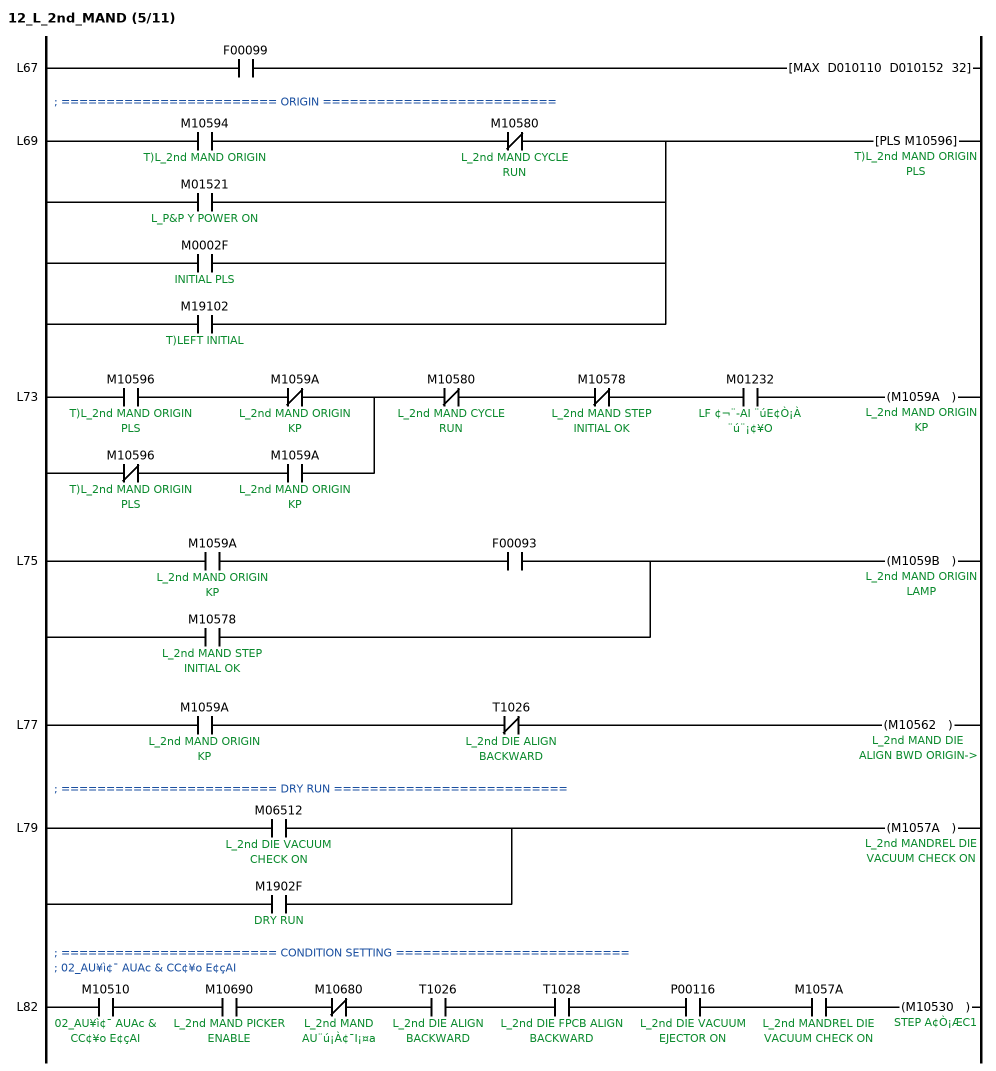
[picture p72: 12_L_2nd_MAND rungs L67-L82]
; L67
LOAD      F00099
MAX       D010110 D010152 32
// ======================== ORIGIN ==========================
; L69
LOAD      M10594	// T)L_2nd MAND ORIGIN
AND NOT   M10580	// L_2nd MAND CYCLE RUN
OR        M01521	// L_P&P Y POWER ON
OR        M0002F	// INITIAL PLS
OR        M19102	// T)LEFT INITIAL
OUTP      M10596	// T)L_2nd MAND ORIGIN PLS
; L73
LOAD      M10596	// T)L_2nd MAND ORIGIN PLS
AND NOT   M1059A	// L_2nd MAND ORIGIN KP
LOAD NOT  M10596	// T)L_2nd MAND ORIGIN PLS
AND       M1059A	// L_2nd MAND ORIGIN KP
OR LOAD
AND NOT   M10580	// L_2nd MAND CYCLE RUN
AND NOT   M10578	// L_2nd MAND STEP INITIAL OK
AND       M01232	// LF ¢¬¨­AI ¨úE¢Ò¡À ¨ú¨¡¢¥O
OUT       M1059A	// L_2nd MAND ORIGIN KP
; L75
LOAD      M1059A	// L_2nd MAND ORIGIN KP
AND       F00093
OR        M10578	// L_2nd MAND STEP INITIAL OK
OUT       M1059B	// L_2nd MAND ORIGIN LAMP
; L77
LOAD      M1059A	// L_2nd MAND ORIGIN KP
AND NOT   T1026	// L_2nd DIE ALIGN BACKWARD
OUT       M10562	// L_2nd MAND DIE ALIGN BWD ORIGIN->
// ======================== DRY RUN ==========================
; L79
LOAD      M06512	// L_2nd DIE VACUUM CHECK ON
OR        M1902F	// DRY RUN
OUT       M1057A	// L_2nd MANDREL DIE VACUUM CHECK ON
// ======================== CONDITION SETTING ==========================
; L82
LOAD      M10510	// 02_AU¥ì¢¯ AUAc & CC¢¥o E¢çAI
AND       M10690	// L_2nd MAND PICKER ENABLE
AND NOT   M10680	// L_2nd MAND AU¨ú¡À¢¯I¡¤a
AND       T1026	// L_2nd DIE ALIGN BACKWARD
AND       T1028	// L_2nd DIE FPCB ALIGN BACKWARD
AND       P00116	// L_2nd DIE VACUUM EJECTOR ON
AND       M1057A	// L_2nd MANDREL DIE VACUUM CHECK ON
OUT       M10530	// STEP A¢Ò¡ÆC1
// output comment: 02_AU¥ì¢¯ AUAc & CC¢¥o E¢çAI

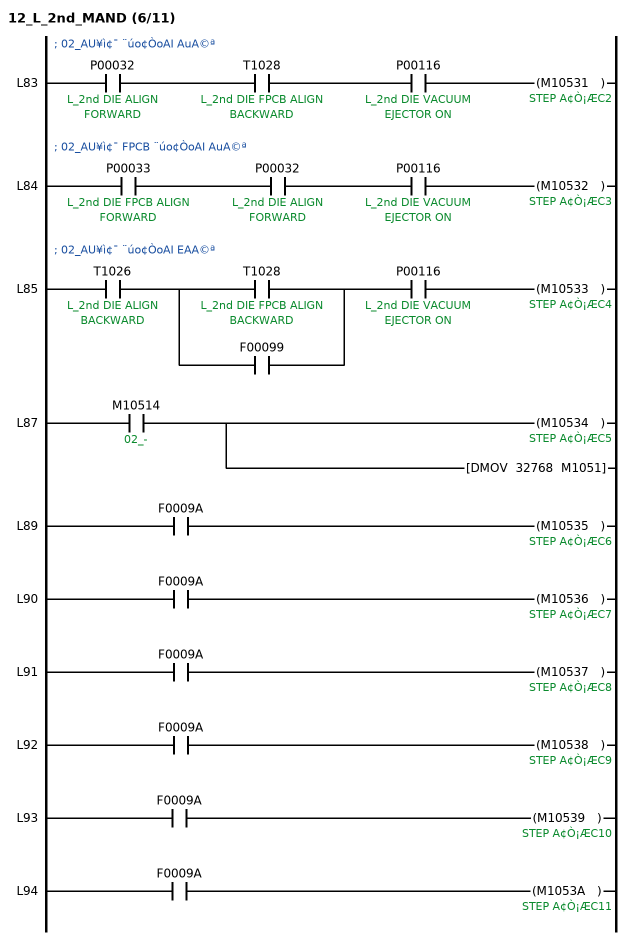
; L83
LOAD      P00032	// L_2nd DIE ALIGN FORWARD
AND       T1028	// L_2nd DIE FPCB ALIGN BACKWARD
AND       P00116	// L_2nd DIE VACUUM EJECTOR ON
OUT       M10531	// STEP A¢Ò¡ÆC2
// output comment: 02_AU¥ì¢¯ ¨úo¢ÒoAI AuA©ª
; L84
LOAD      P00033	// L_2nd DIE FPCB ALIGN FORWARD
AND       P00032	// L_2nd DIE ALIGN FORWARD
AND       P00116	// L_2nd DIE VACUUM EJECTOR ON
OUT       M10532	// STEP A¢Ò¡ÆC3
// output comment: 02_AU¥ì¢¯ FPCB ¨úo¢ÒoAI AuA©ª
; L85
LOAD      T1026	// L_2nd DIE ALIGN BACKWARD
LOAD      T1028	// L_2nd DIE FPCB ALIGN BACKWARD
OR        F00099
AND LOAD
AND       P00116	// L_2nd DIE VACUUM EJECTOR ON
OUT       M10533	// STEP A¢Ò¡ÆC4
// output comment: 02_AU¥ì¢¯ ¨úo¢ÒoAI EAA©ª
; L87
LOAD      M10514	// 02_-
OUT       M10534	// STEP A¢Ò¡ÆC5
DMOV      32768 M1051
; L89
LOAD      F0009A
OUT       M10535	// STEP A¢Ò¡ÆC6
; L90
LOAD      F0009A
OUT       M10536	// STEP A¢Ò¡ÆC7
; L91
LOAD      F0009A
OUT       M10537	// STEP A¢Ò¡ÆC8
; L92
LOAD      F0009A
OUT       M10538	// STEP A¢Ò¡ÆC9
; L93
LOAD      F0009A
OUT       M10539	// STEP A¢Ò¡ÆC10
; L94
LOAD      F0009A
OUT       M1053A	// STEP A¢Ò¡ÆC11

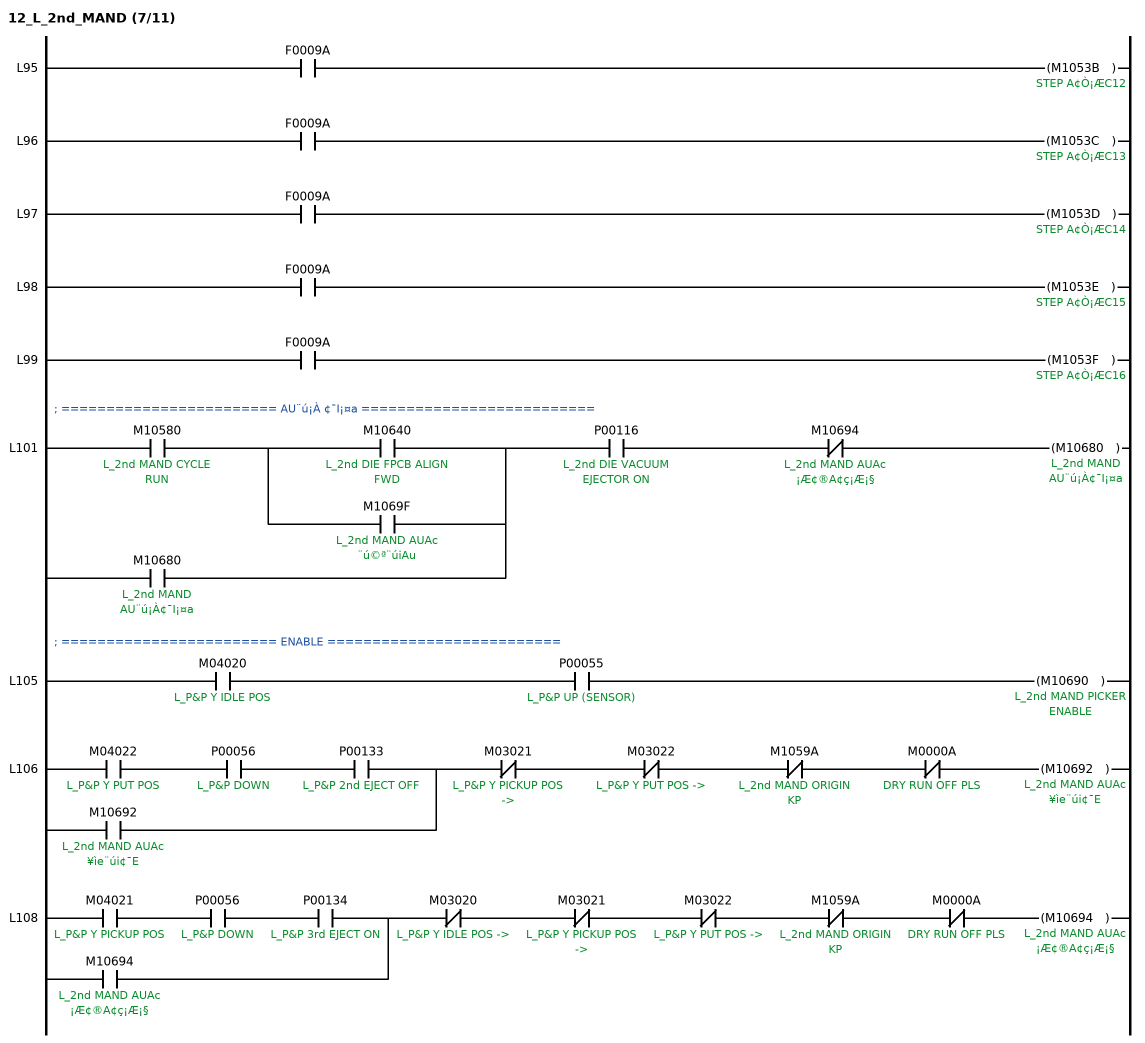
; L95
LOAD      F0009A
OUT       M1053B	// STEP A¢Ò¡ÆC12
; L96
LOAD      F0009A
OUT       M1053C	// STEP A¢Ò¡ÆC13
; L97
LOAD      F0009A
OUT       M1053D	// STEP A¢Ò¡ÆC14
; L98
LOAD      F0009A
OUT       M1053E	// STEP A¢Ò¡ÆC15
; L99
LOAD      F0009A
OUT       M1053F	// STEP A¢Ò¡ÆC16
// ======================== AU¨ú¡À ¢¯I¡¤a ==========================
; L101
LOAD      M10580	// L_2nd MAND CYCLE RUN
LOAD      M10640	// L_2nd DIE FPCB ALIGN FWD
OR        M1069F	// L_2nd MAND AUAc ¨ú©ª¨úiAu
AND LOAD
OR        M10680	// L_2nd MAND AU¨ú¡À¢¯I¡¤a
AND       P00116	// L_2nd DIE VACUUM EJECTOR ON
AND NOT   M10694	// L_2nd MAND AUAc ¡Æ¢®A¢ç¡Æ¡§
OUT       M10680	// L_2nd MAND AU¨ú¡À¢¯I¡¤a
// ======================== ENABLE ==========================
; L105
LOAD      M04020	// L_P&P Y IDLE POS
AND       P00055	// L_P&P UP (SENSOR)
OUT       M10690	// L_2nd MAND PICKER ENABLE
; L106
LOAD      M04022	// L_P&P Y PUT POS
AND       P00056	// L_P&P DOWN
AND       P00133	// L_P&P 2nd EJECT OFF
OR        M10692	// L_2nd MAND AUAc ¥ìe¨úi¢¯E
AND NOT   M03021	// L_P&P Y PICKUP POS ->
AND NOT   M03022	// L_P&P Y PUT POS ->
AND NOT   M1059A	// L_2nd MAND ORIGIN KP
AND NOT   M0000A	// DRY RUN OFF PLS
OUT       M10692	// L_2nd MAND AUAc ¥ìe¨úi¢¯E
; L108
LOAD      M04021	// L_P&P Y PICKUP POS
AND       P00056	// L_P&P DOWN
AND       P00134	// L_P&P 3rd EJECT ON
OR        M10694	// L_2nd MAND AUAc ¡Æ¢®A¢ç¡Æ¡§
AND NOT   M03020	// L_P&P Y IDLE POS ->
AND NOT   M03021	// L_P&P Y PICKUP POS ->
AND NOT   M03022	// L_P&P Y PUT POS ->
AND NOT   M1059A	// L_2nd MAND ORIGIN KP
AND NOT   M0000A	// DRY RUN OFF PLS
OUT       M10694	// L_2nd MAND AUAc ¡Æ¢®A¢ç¡Æ¡§

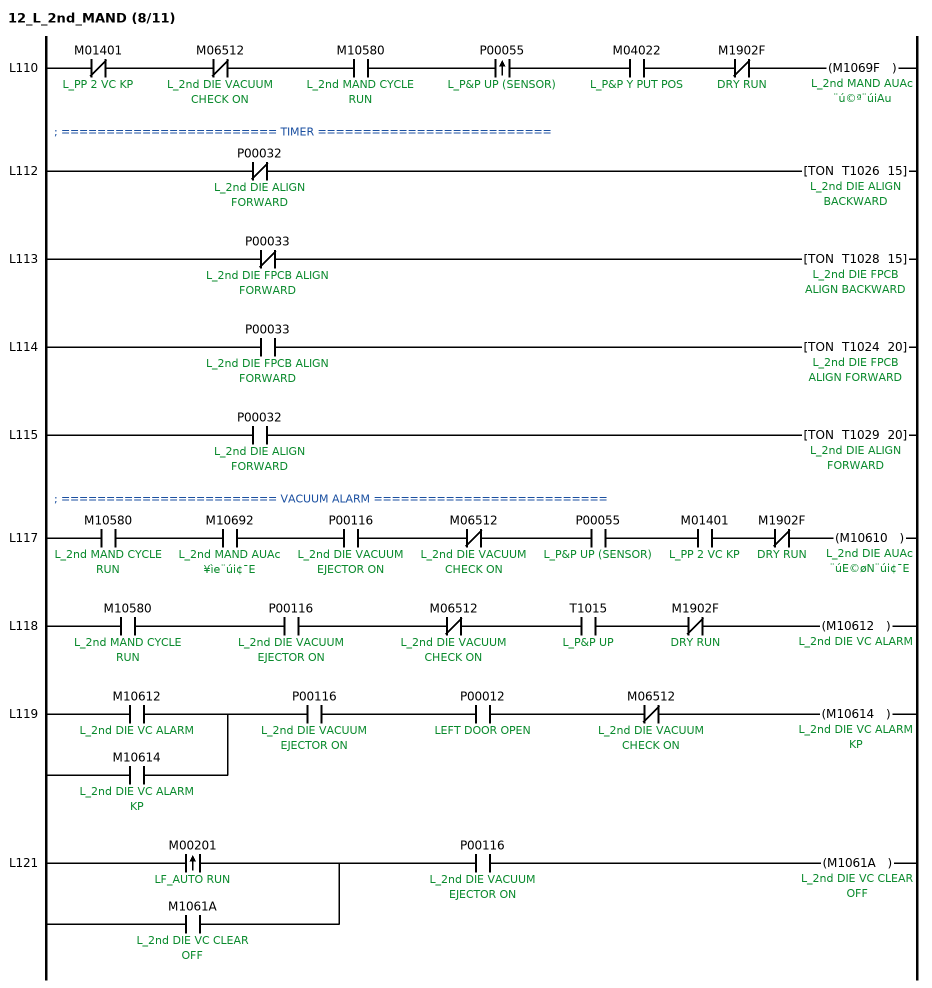
; L110
LOAD NOT  M01401	// L_PP 2 VC KP
AND NOT   M06512	// L_2nd DIE VACUUM CHECK ON
AND       M10580	// L_2nd MAND CYCLE RUN
ANDP      P00055	// L_P&P UP (SENSOR)
AND       M04022	// L_P&P Y PUT POS
AND NOT   M1902F	// DRY RUN
OUT       M1069F	// L_2nd MAND AUAc ¨ú©ª¨úiAu
// ======================== TIMER ==========================
; L112
LOAD NOT  P00032	// L_2nd DIE ALIGN FORWARD
TON       T1026 15	// L_2nd DIE ALIGN BACKWARD
; L113
LOAD NOT  P00033	// L_2nd DIE FPCB ALIGN FORWARD
TON       T1028 15	// L_2nd DIE FPCB ALIGN BACKWARD
; L114
LOAD      P00033	// L_2nd DIE FPCB ALIGN FORWARD
TON       T1024 20	// L_2nd DIE FPCB ALIGN FORWARD
; L115
LOAD      P00032	// L_2nd DIE ALIGN FORWARD
TON       T1029 20	// L_2nd DIE ALIGN FORWARD
// ======================== VACUUM ALARM ==========================
; L117
LOAD      M10580	// L_2nd MAND CYCLE RUN
AND       M10692	// L_2nd MAND AUAc ¥ìe¨úi¢¯E
AND       P00116	// L_2nd DIE VACUUM EJECTOR ON
AND NOT   M06512	// L_2nd DIE VACUUM CHECK ON
AND       P00055	// L_P&P UP (SENSOR)
AND       M01401	// L_PP 2 VC KP
AND NOT   M1902F	// DRY RUN
OUT       M10610	// L_2nd DIE AUAc ¨úE©øN¨úi¢¯E
; L118
LOAD      M10580	// L_2nd MAND CYCLE RUN
AND       P00116	// L_2nd DIE VACUUM EJECTOR ON
AND NOT   M06512	// L_2nd DIE VACUUM CHECK ON
AND       T1015	// L_P&P UP
AND NOT   M1902F	// DRY RUN
OUT       M10612	// L_2nd DIE VC ALARM
; L119
LOAD      M10612	// L_2nd DIE VC ALARM
OR        M10614	// L_2nd DIE VC ALARM KP
AND       P00116	// L_2nd DIE VACUUM EJECTOR ON
AND       P00012	// LEFT DOOR OPEN
AND NOT   M06512	// L_2nd DIE VACUUM CHECK ON
OUT       M10614	// L_2nd DIE VC ALARM KP
; L121
LOADP     M00201	// LF_AUTO RUN
OR        M1061A	// L_2nd DIE VC CLEAR OFF
AND       P00116	// L_2nd DIE VACUUM EJECTOR ON
OUT       M1061A	// L_2nd DIE VC CLEAR OFF

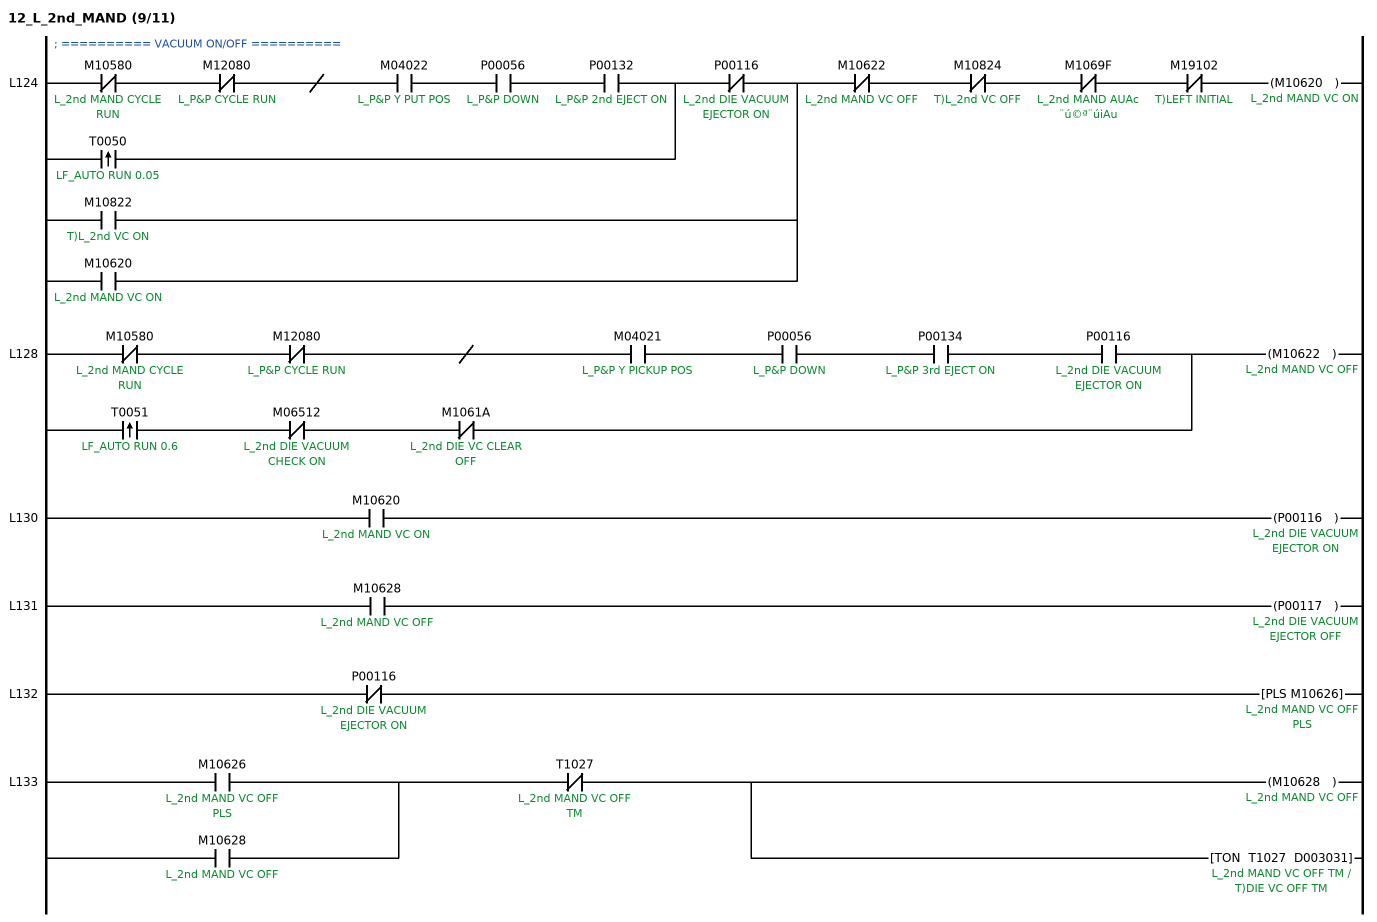
// ========== VACUUM ON/OFF ==========
; L124
LOAD NOT  M10580	// L_2nd MAND CYCLE RUN
AND NOT   M12080	// L_P&P CYCLE RUN
NOT
AND       M04022	// L_P&P Y PUT POS
AND       P00056	// L_P&P DOWN
AND       P00132	// L_P&P 2nd EJECT ON
ORP       T0050	// LF_AUTO RUN 0.05
AND NOT   P00116	// L_2nd DIE VACUUM EJECTOR ON
OR        M10822	// T)L_2nd VC ON
OR        M10620	// L_2nd MAND VC ON
AND NOT   M10622	// L_2nd MAND VC OFF
AND NOT   M10824	// T)L_2nd VC OFF
AND NOT   M1069F	// L_2nd MAND AUAc ¨ú©ª¨úiAu
AND NOT   M19102	// T)LEFT INITIAL
OUT       M10620	// L_2nd MAND VC ON
; L128
LOAD NOT  M10580	// L_2nd MAND CYCLE RUN
AND NOT   M12080	// L_P&P CYCLE RUN
NOT
AND       M04021	// L_P&P Y PICKUP POS
AND       P00056	// L_P&P DOWN
AND       P00134	// L_P&P 3rd EJECT ON
AND       P00116	// L_2nd DIE VACUUM EJECTOR ON
LOADP     T0051	// LF_AUTO RUN 0.6
AND NOT   M06512	// L_2nd DIE VACUUM CHECK ON
AND NOT   M1061A	// L_2nd DIE VC CLEAR OFF
OR LOAD
OUT       M10622	// L_2nd MAND VC OFF
; L130
LOAD      M10620	// L_2nd MAND VC ON
OUT       P00116	// L_2nd DIE VACUUM EJECTOR ON
; L131
LOAD      M10628	// L_2nd MAND VC OFF
OUT       P00117	// L_2nd DIE VACUUM EJECTOR OFF
; L132
LOAD NOT  P00116	// L_2nd DIE VACUUM EJECTOR ON
OUTP      M10626	// L_2nd MAND VC OFF PLS
; L133
LOAD      M10626	// L_2nd MAND VC OFF PLS
OR        M10628	// L_2nd MAND VC OFF
AND NOT   T1027	// L_2nd MAND VC OFF TM
OUT       M10628	// L_2nd MAND VC OFF
TON       T1027 D003031	// L_2nd MAND VC OFF TM / T)DIE VC OFF TM

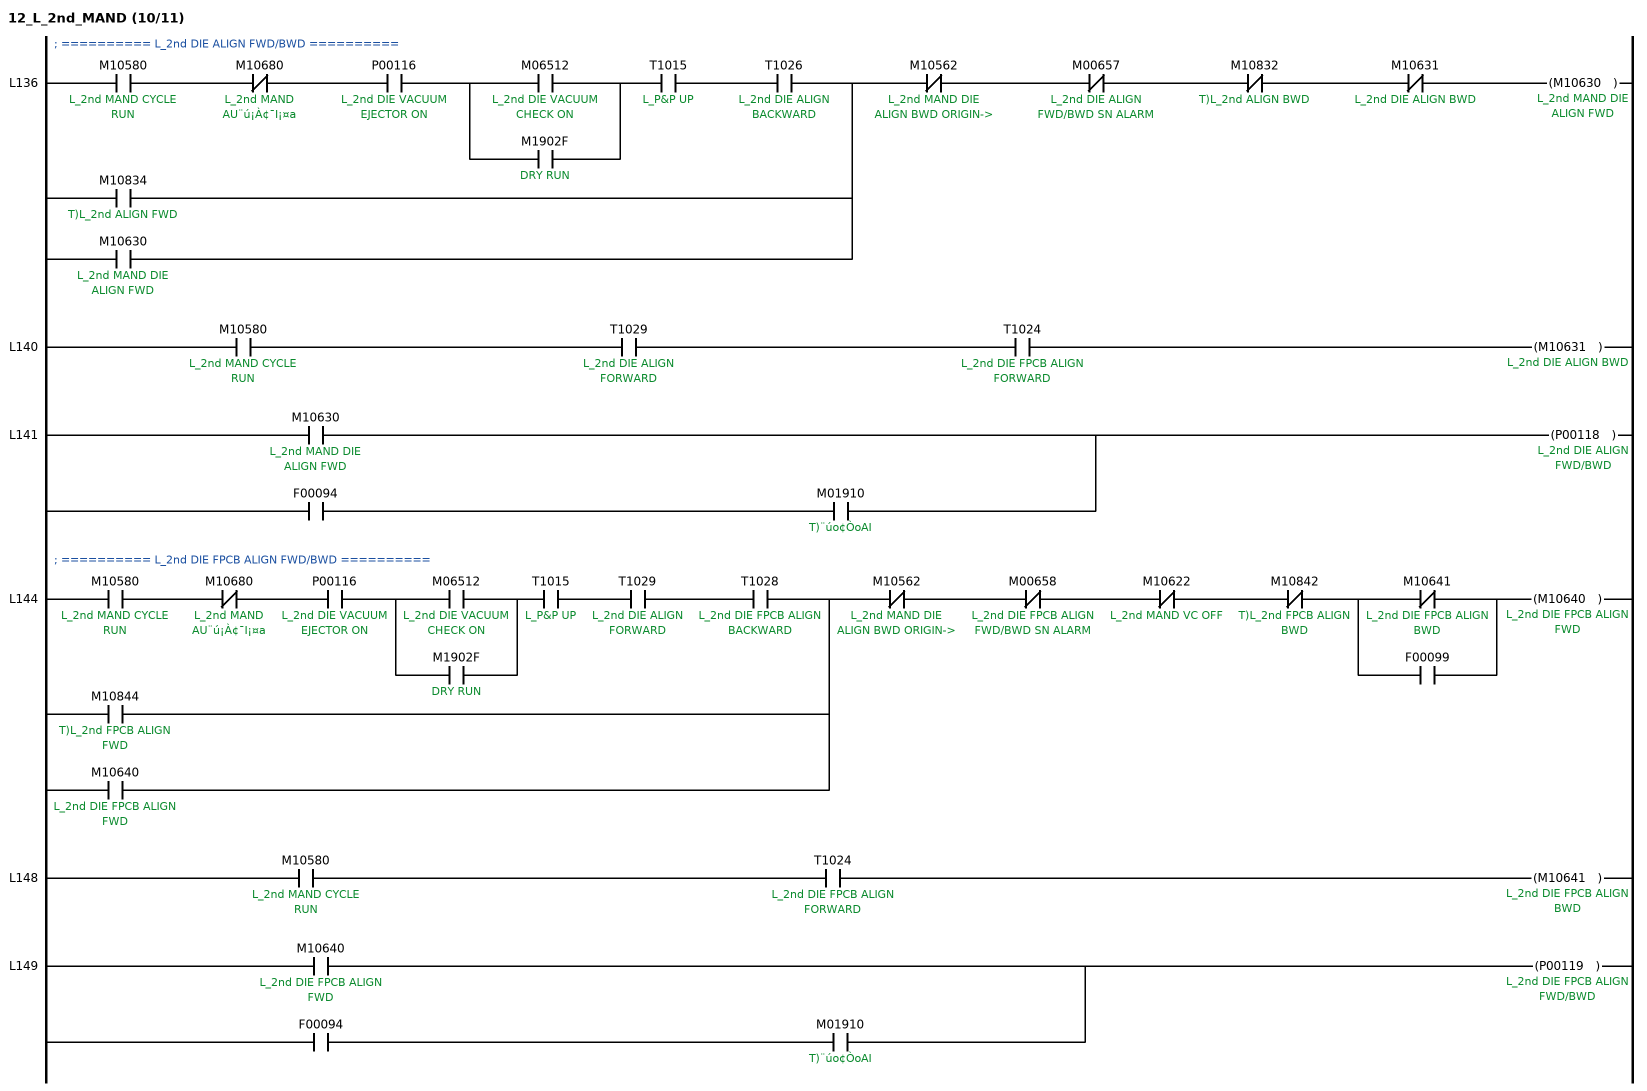
// ========== L_2nd DIE ALIGN FWD/BWD ==========
; L136
LOAD      M10580	// L_2nd MAND CYCLE RUN
AND NOT   M10680	// L_2nd MAND AU¨ú¡À¢¯I¡¤a
AND       P00116	// L_2nd DIE VACUUM EJECTOR ON
LOAD      M06512	// L_2nd DIE VACUUM CHECK ON
OR        M1902F	// DRY RUN
AND LOAD
AND       T1015	// L_P&P UP
AND       T1026	// L_2nd DIE ALIGN BACKWARD
OR        M10834	// T)L_2nd ALIGN FWD
OR        M10630	// L_2nd MAND DIE ALIGN FWD
AND NOT   M10562	// L_2nd MAND DIE ALIGN BWD ORIGIN->
AND NOT   M00657	// L_2nd DIE ALIGN FWD/BWD SN ALARM
AND NOT   M10832	// T)L_2nd ALIGN BWD
AND NOT   M10631	// L_2nd DIE ALIGN BWD
OUT       M10630	// L_2nd MAND DIE ALIGN FWD
; L140
LOAD      M10580	// L_2nd MAND CYCLE RUN
AND       T1029	// L_2nd DIE ALIGN FORWARD
AND       T1024	// L_2nd DIE FPCB ALIGN FORWARD
OUT       M10631	// L_2nd DIE ALIGN BWD
; L141
LOAD      M10630	// L_2nd MAND DIE ALIGN FWD
LOAD      F00094
AND       M01910	// T)¨úo¢ÒoAI
OR LOAD
OUT       P00118	// L_2nd DIE ALIGN FWD/BWD
// ========== L_2nd DIE FPCB ALIGN FWD/BWD ==========
; L144
LOAD      M10580	// L_2nd MAND CYCLE RUN
AND NOT   M10680	// L_2nd MAND AU¨ú¡À¢¯I¡¤a
AND       P00116	// L_2nd DIE VACUUM EJECTOR ON
LOAD      M06512	// L_2nd DIE VACUUM CHECK ON
OR        M1902F	// DRY RUN
AND LOAD
AND       T1015	// L_P&P UP
AND       T1029	// L_2nd DIE ALIGN FORWARD
AND       T1028	// L_2nd DIE FPCB ALIGN BACKWARD
OR        M10844	// T)L_2nd FPCB ALIGN FWD
OR        M10640	// L_2nd DIE FPCB ALIGN FWD
AND NOT   M10562	// L_2nd MAND DIE ALIGN BWD ORIGIN->
AND NOT   M00658	// L_2nd DIE FPCB ALIGN FWD/BWD SN ALARM
AND NOT   M10622	// L_2nd MAND VC OFF
AND NOT   M10842	// T)L_2nd FPCB ALIGN BWD
LOAD NOT  M10641	// L_2nd DIE FPCB ALIGN BWD
OR        F00099
AND LOAD
OUT       M10640	// L_2nd DIE FPCB ALIGN FWD
; L148
LOAD      M10580	// L_2nd MAND CYCLE RUN
AND       T1024	// L_2nd DIE FPCB ALIGN FORWARD
OUT       M10641	// L_2nd DIE FPCB ALIGN BWD
; L149
LOAD      M10640	// L_2nd DIE FPCB ALIGN FWD
LOAD      F00094
AND       M01910	// T)¨úo¢ÒoAI
OR LOAD
OUT       P00119	// L_2nd DIE FPCB ALIGN FWD/BWD

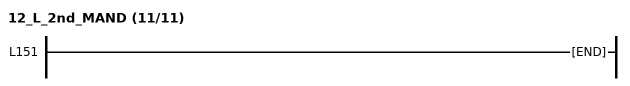
; L151
END

PROGRAM 13_L_3rd_MAND (task: ¨ö¨¬A¥ì CA¡¤I¡¾¡¿¡¤¡Í)

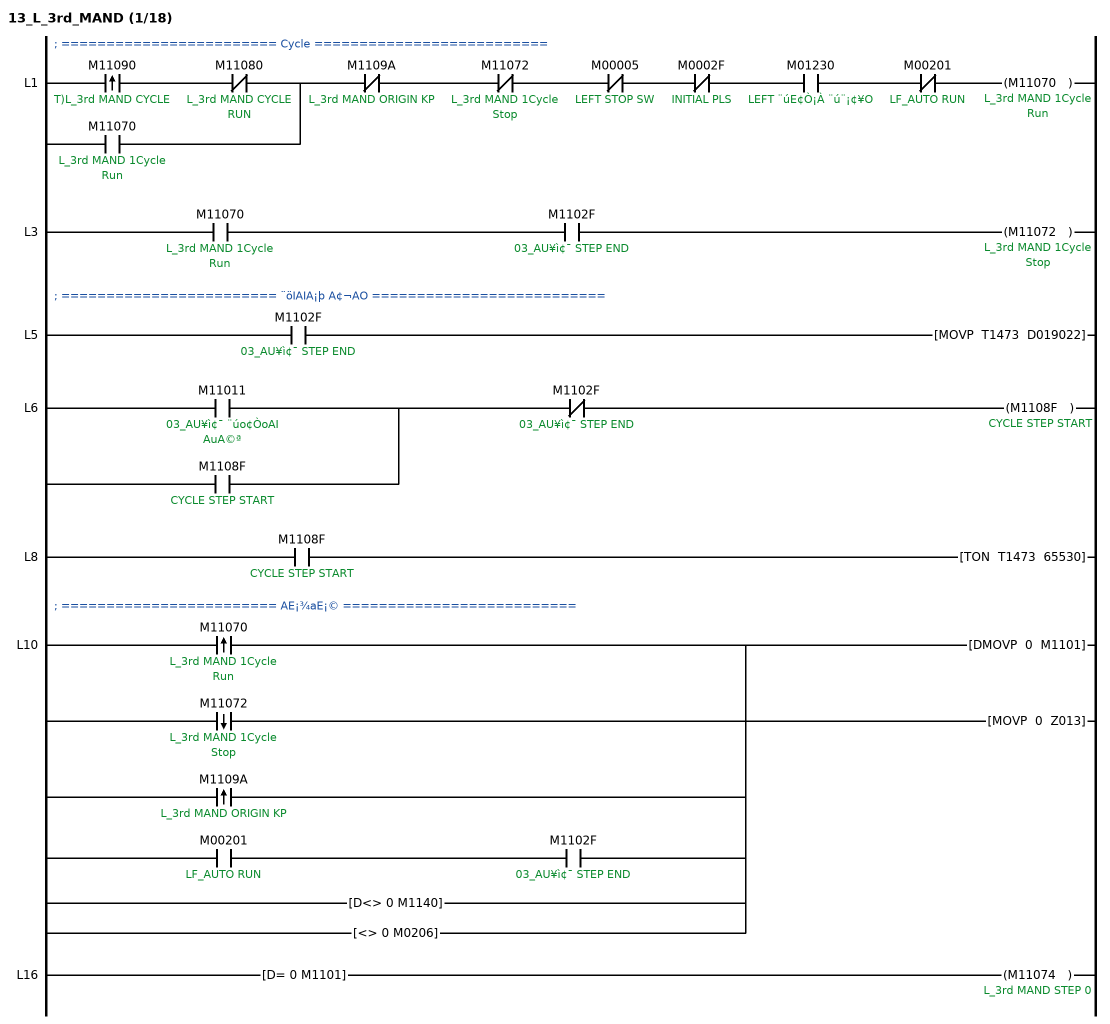
// ======================== Cycle ==========================
; L1
LOADP     M11090	// T)L_3rd MAND CYCLE
AND NOT   M11080	// L_3rd MAND CYCLE RUN
OR        M11070	// L_3rd MAND 1Cycle Run
AND NOT   M1109A	// L_3rd MAND ORIGIN KP
AND NOT   M11072	// L_3rd MAND 1Cycle Stop
AND NOT   M00005	// LEFT STOP SW
AND NOT   M0002F	// INITIAL PLS
AND       M01230	// LEFT ¨úE¢Ò¡À ¨ú¨¡¢¥O
AND NOT   M00201	// LF_AUTO RUN
OUT       M11070	// L_3rd MAND 1Cycle Run
; L3
LOAD      M11070	// L_3rd MAND 1Cycle Run
AND       M1102F	// 03_AU¥ì¢¯ STEP END
OUT       M11072	// L_3rd MAND 1Cycle Stop
// ======================== ¨öIAIA¡þ A¢¬AO ==========================
; L5
LOAD      M1102F	// 03_AU¥ì¢¯ STEP END
MOVP      T1473 D019022
; L6
LOAD      M11011	// 03_AU¥ì¢¯ ¨úo¢ÒoAI AuA©ª
OR        M1108F	// CYCLE STEP START
AND NOT   M1102F	// 03_AU¥ì¢¯ STEP END
OUT       M1108F	// CYCLE STEP START
; L8
LOAD      M1108F	// CYCLE STEP START
TON       T1473 65530
// ======================== AE¡¾aE¡© ==========================
; L10
LOADP     M11070	// L_3rd MAND 1Cycle Run
ORN       M11072	// L_3rd MAND 1Cycle Stop
ORP       M1109A	// L_3rd MAND ORIGIN KP
LOAD      M00201	// LF_AUTO RUN
AND       M1102F	// 03_AU¥ì¢¯ STEP END
OR LOAD
ORD<>     0 M1140
OR<>      0 M0206
DMOVP     0 M1101
MOVP      0 Z013
; L16
LOADD=    0 M1101
OUT       M11074	// L_3rd MAND STEP 0

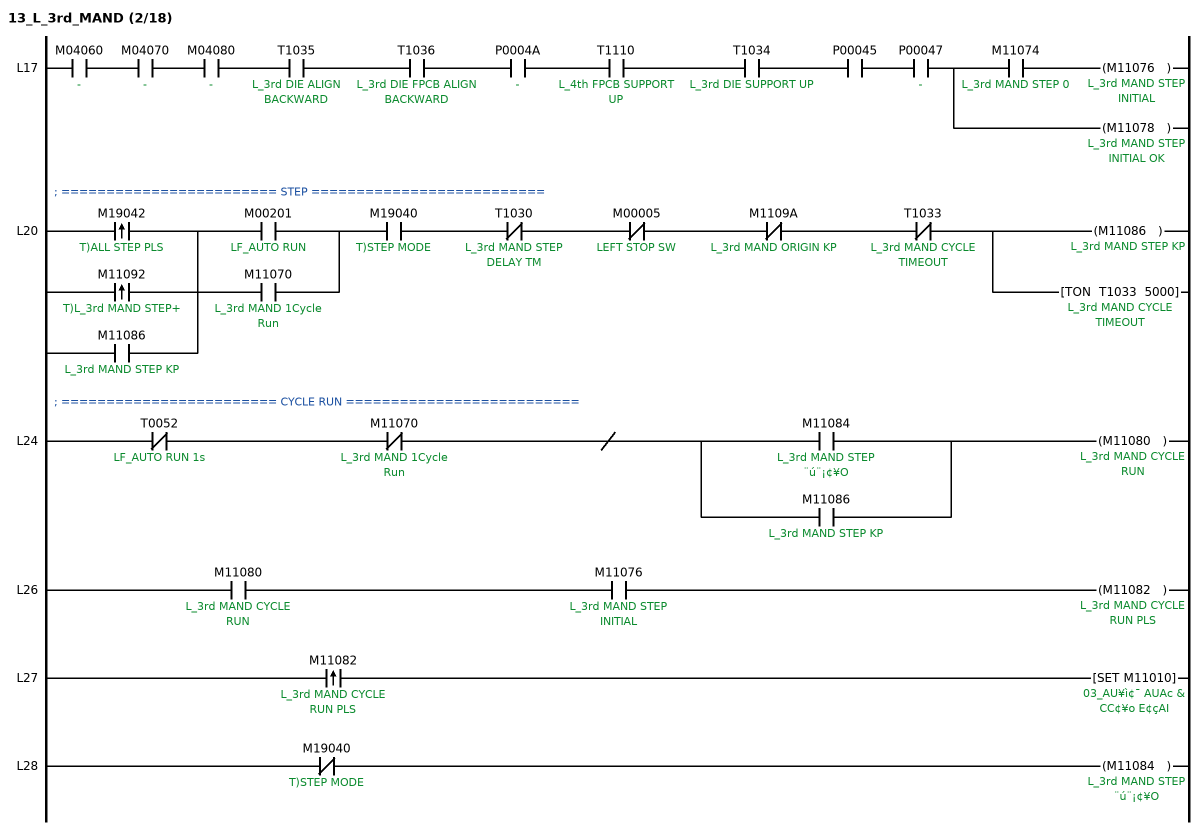
; L17
LOAD      M04060	// -
AND       M04070	// -
AND       M04080	// -
AND       T1035	// L_3rd DIE ALIGN BACKWARD
AND       T1036	// L_3rd DIE FPCB ALIGN BACKWARD
AND       P0004A	// -
AND       T1110	// L_4th FPCB SUPPORT UP
AND       T1034	// L_3rd DIE SUPPORT UP
AND       P00045
AND       P00047	// -
MPUSH
AND       M11074	// L_3rd MAND STEP 0
OUT       M11076	// L_3rd MAND STEP INITIAL
MPOP
OUT       M11078	// L_3rd MAND STEP INITIAL OK
// ======================== STEP ==========================
; L20
LOADP     M19042	// T)ALL STEP PLS
ORP       M11092	// T)L_3rd MAND STEP+
OR        M11086	// L_3rd MAND STEP KP
LOAD      M00201	// LF_AUTO RUN
OR        M11070	// L_3rd MAND 1Cycle Run
AND LOAD
AND       M19040	// T)STEP MODE
AND NOT   T1030	// L_3rd MAND STEP DELAY TM
AND NOT   M00005	// LEFT STOP SW
AND NOT   M1109A	// L_3rd MAND ORIGIN KP
AND NOT   T1033	// L_3rd MAND CYCLE TIMEOUT
OUT       M11086	// L_3rd MAND STEP KP
TON       T1033 5000	// L_3rd MAND CYCLE TIMEOUT
// ======================== CYCLE RUN ==========================
; L24
LOAD NOT  T0052	// LF_AUTO RUN 1s
AND NOT   M11070	// L_3rd MAND 1Cycle Run
NOT
LOAD      M11084	// L_3rd MAND STEP ¨ú¨¡¢¥O
OR        M11086	// L_3rd MAND STEP KP
AND LOAD
OUT       M11080	// L_3rd MAND CYCLE RUN
; L26
LOAD      M11080	// L_3rd MAND CYCLE RUN
AND       M11076	// L_3rd MAND STEP INITIAL
OUT       M11082	// L_3rd MAND CYCLE RUN PLS
; L27
LOADP     M11082	// L_3rd MAND CYCLE RUN PLS
SET       M11010	// 03_AU¥ì¢¯ AUAc & CC¢¥o E¢çAI
; L28
LOAD NOT  M19040	// T)STEP MODE
OUT       M11084	// L_3rd MAND STEP ¨ú¨¡¢¥O

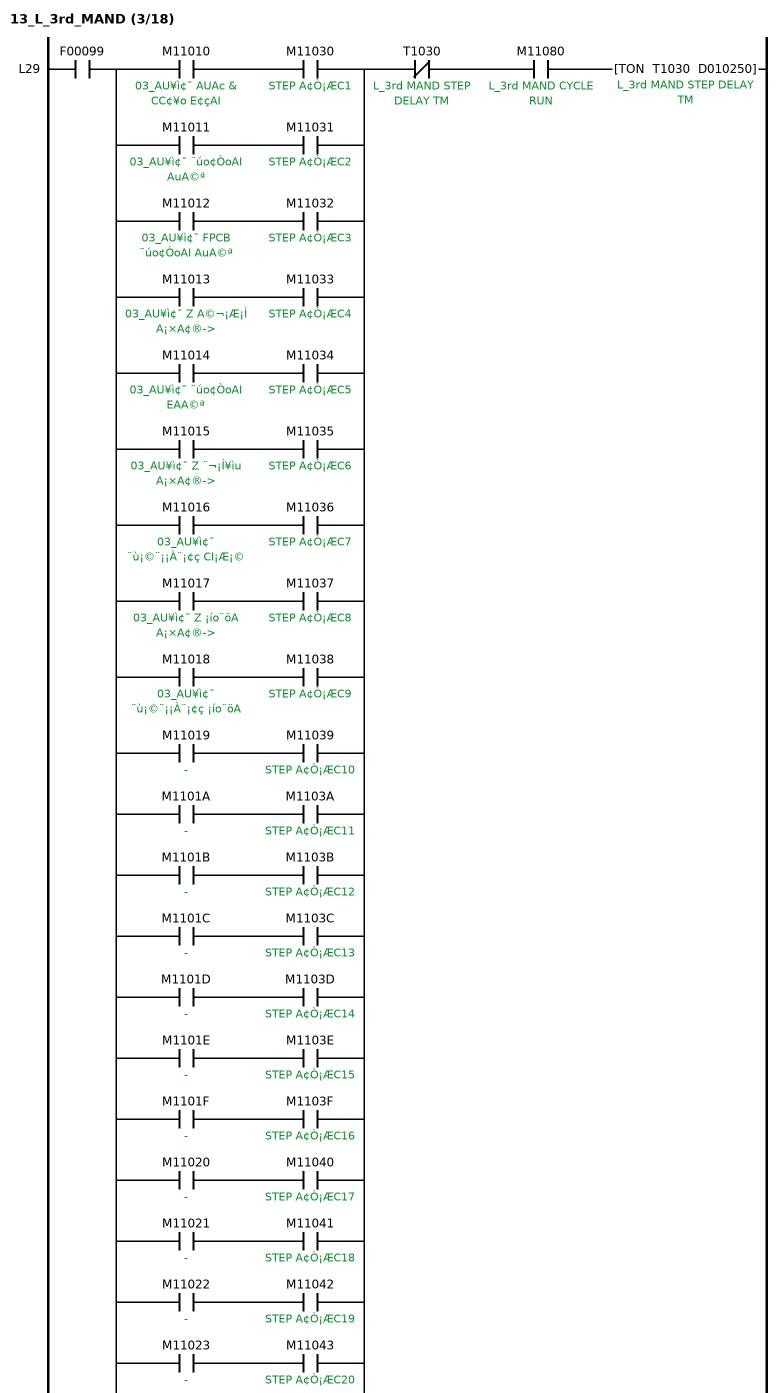

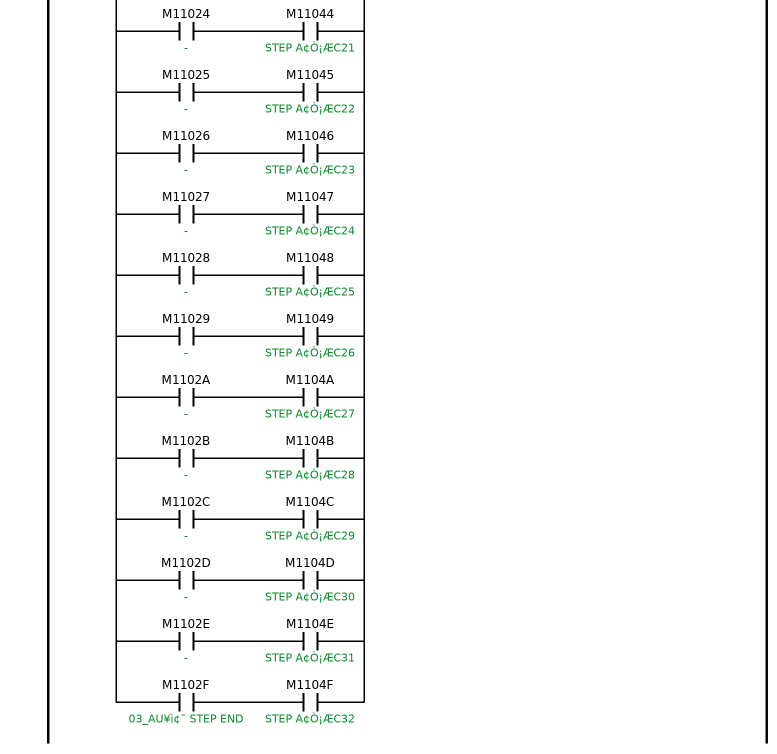
; L29
LOAD      F00099
LOAD      M11010	// 03_AU¥ì¢¯ AUAc & CC¢¥o E¢çAI
AND       M11030	// STEP A¢Ò¡ÆC1
LOAD      M11011	// 03_AU¥ì¢¯ ¨úo¢ÒoAI AuA©ª
AND       M11031	// STEP A¢Ò¡ÆC2
OR LOAD
LOAD      M11012	// 03_AU¥ì¢¯ FPCB ¨úo¢ÒoAI AuA©ª
AND       M11032	// STEP A¢Ò¡ÆC3
OR LOAD
LOAD      M11013	// 03_AU¥ì¢¯ Z A©¬¡Æ¡Ì A¡×A¢®->
AND       M11033	// STEP A¢Ò¡ÆC4
OR LOAD
LOAD      M11014	// 03_AU¥ì¢¯ ¨úo¢ÒoAI EAA©ª
AND       M11034	// STEP A¢Ò¡ÆC5
OR LOAD
LOAD      M11015	// 03_AU¥ì¢¯ Z ¨¬¡Í¥ìu A¡×A¢®->
AND       M11035	// STEP A¢Ò¡ÆC6
OR LOAD
LOAD      M11016	// 03_AU¥ì¢¯ ¨ù¡©¨¡¡À¨¡¢ç CI¡Æ¡©
AND       M11036	// STEP A¢Ò¡ÆC7
OR LOAD
LOAD      M11017	// 03_AU¥ì¢¯ Z ¡ío¨öA A¡×A¢®->
AND       M11037	// STEP A¢Ò¡ÆC8
OR LOAD
LOAD      M11018	// 03_AU¥ì¢¯ ¨ù¡©¨¡¡À¨¡¢ç ¡ío¨öA
AND       M11038	// STEP A¢Ò¡ÆC9
OR LOAD
LOAD      M11019	// -
AND       M11039	// STEP A¢Ò¡ÆC10
OR LOAD
LOAD      M1101A	// -
AND       M1103A	// STEP A¢Ò¡ÆC11
OR LOAD
LOAD      M1101B	// -
AND       M1103B	// STEP A¢Ò¡ÆC12
OR LOAD
LOAD      M1101C	// -
AND       M1103C	// STEP A¢Ò¡ÆC13
OR LOAD
LOAD      M1101D	// -
AND       M1103D	// STEP A¢Ò¡ÆC14
OR LOAD
LOAD      M1101E	// -
AND       M1103E	// STEP A¢Ò¡ÆC15
OR LOAD
LOAD      M1101F	// -
AND       M1103F	// STEP A¢Ò¡ÆC16
OR LOAD
LOAD      M11020	// -
AND       M11040	// STEP A¢Ò¡ÆC17
OR LOAD
LOAD      M11021	// -
AND       M11041	// STEP A¢Ò¡ÆC18
OR LOAD
LOAD      M11022	// -
AND       M11042	// STEP A¢Ò¡ÆC19
OR LOAD
LOAD      M11023	// -
AND       M11043	// STEP A¢Ò¡ÆC20
OR LOAD
LOAD      M11024	// -
AND       M11044	// STEP A¢Ò¡ÆC21
OR LOAD
LOAD      M11025	// -
AND       M11045	// STEP A¢Ò¡ÆC22
OR LOAD
LOAD      M11026	// -
AND       M11046	// STEP A¢Ò¡ÆC23
OR LOAD
LOAD      M11027	// -
AND       M11047	// STEP A¢Ò¡ÆC24
OR LOAD
LOAD      M11028	// -
AND       M11048	// STEP A¢Ò¡ÆC25
OR LOAD
LOAD      M11029	// -
AND       M11049	// STEP A¢Ò¡ÆC26
OR LOAD
LOAD      M1102A	// -
AND       M1104A	// STEP A¢Ò¡ÆC27
OR LOAD
LOAD      M1102B	// -
AND       M1104B	// STEP A¢Ò¡ÆC28
OR LOAD
LOAD      M1102C	// -
AND       M1104C	// STEP A¢Ò¡ÆC29
OR LOAD
LOAD      M1102D	// -
AND       M1104D	// STEP A¢Ò¡ÆC30
OR LOAD
LOAD      M1102E	// -
AND       M1104E	// STEP A¢Ò¡ÆC31
OR LOAD
LOAD      M1102F	// 03_AU¥ì¢¯ STEP END
AND       M1104F	// STEP A¢Ò¡ÆC32
OR LOAD
AND LOAD
AND NOT   T1030	// L_3rd MAND STEP DELAY TM
AND       M11080	// L_3rd MAND CYCLE RUN
TON       T1030 D010250	// L_3rd MAND STEP DELAY TM

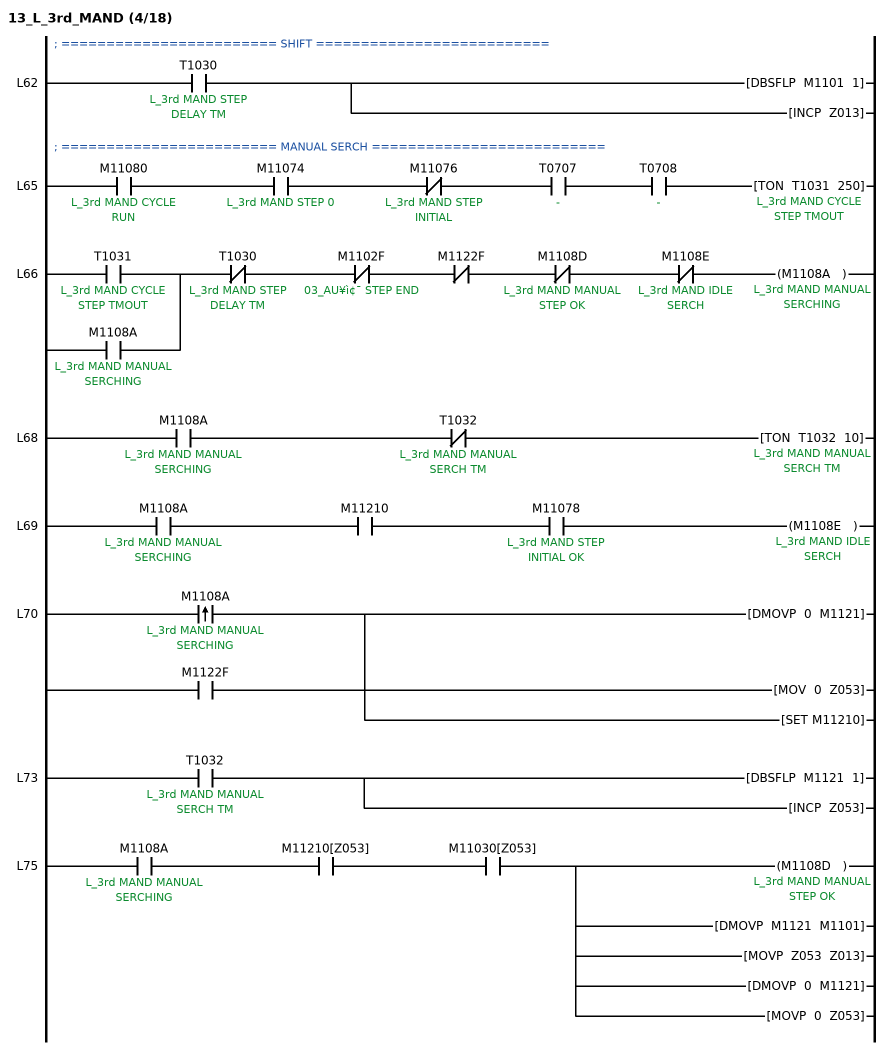
// ======================== SHIFT ==========================
; L62
LOAD      T1030	// L_3rd MAND STEP DELAY TM
DBSFLP    M1101 1
INCP      Z013
// ======================== MANUAL SERCH ==========================
; L65
LOAD      M11080	// L_3rd MAND CYCLE RUN
AND       M11074	// L_3rd MAND STEP 0
AND NOT   M11076	// L_3rd MAND STEP INITIAL
AND       T0707	// -
AND       T0708	// -
TON       T1031 250	// L_3rd MAND CYCLE STEP TMOUT
; L66
LOAD      T1031	// L_3rd MAND CYCLE STEP TMOUT
OR        M1108A	// L_3rd MAND MANUAL SERCHING
AND NOT   T1030	// L_3rd MAND STEP DELAY TM
AND NOT   M1102F	// 03_AU¥ì¢¯ STEP END
AND NOT   M1122F
AND NOT   M1108D	// L_3rd MAND MANUAL STEP OK
AND NOT   M1108E	// L_3rd MAND IDLE SERCH
OUT       M1108A	// L_3rd MAND MANUAL SERCHING
; L68
LOAD      M1108A	// L_3rd MAND MANUAL SERCHING
AND NOT   T1032	// L_3rd MAND MANUAL SERCH TM
TON       T1032 10	// L_3rd MAND MANUAL SERCH TM
; L69
LOAD      M1108A	// L_3rd MAND MANUAL SERCHING
AND       M11210
AND       M11078	// L_3rd MAND STEP INITIAL OK
OUT       M1108E	// L_3rd MAND IDLE SERCH
; L70
LOADP     M1108A	// L_3rd MAND MANUAL SERCHING
OR        M1122F
DMOVP     0 M1121
MOV       0 Z053
SET       M11210
; L73
LOAD      T1032	// L_3rd MAND MANUAL SERCH TM
DBSFLP    M1121 1
INCP      Z053
; L75
LOAD      M1108A	// L_3rd MAND MANUAL SERCHING
AND       M11210[Z053]
AND       M11030[Z053]
OUT       M1108D	// L_3rd MAND MANUAL STEP OK
DMOVP     M1121 M1101
MOVP      Z053 Z013
DMOVP     0 M1121
MOVP      0 Z053

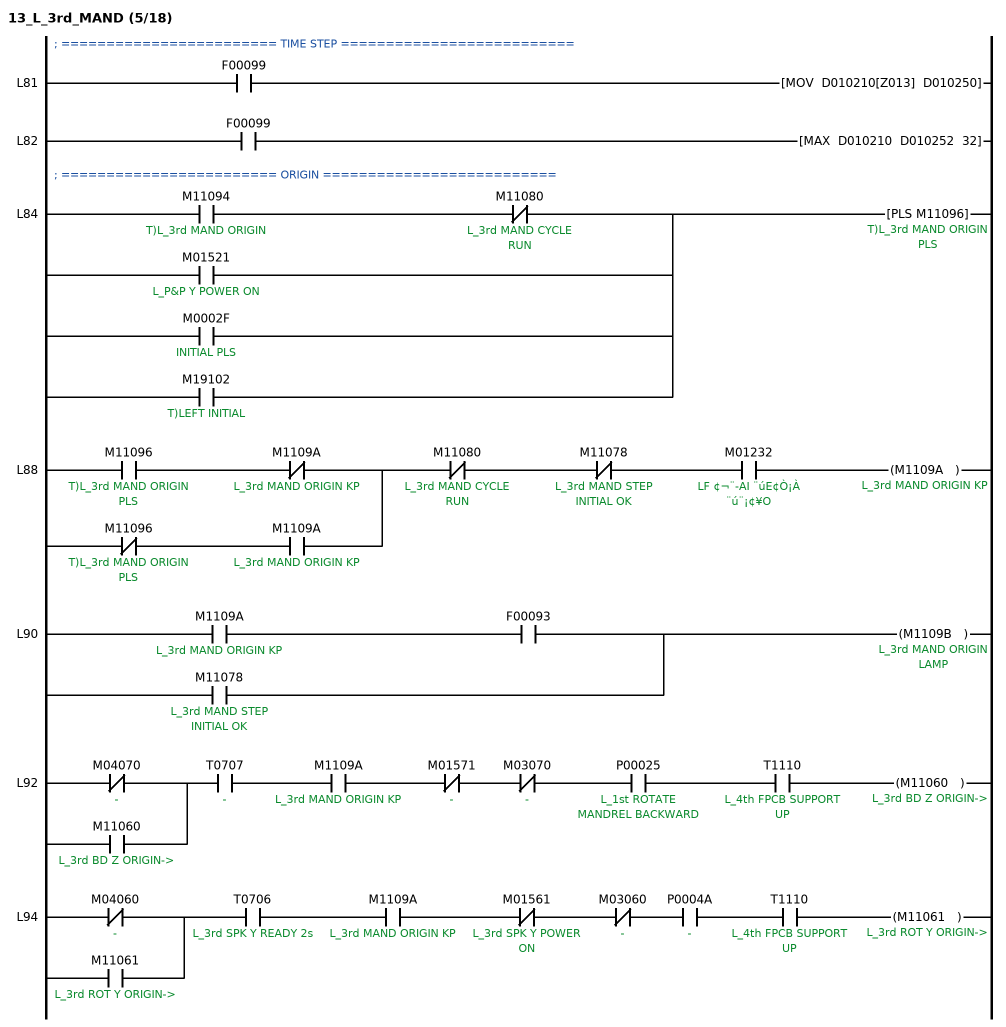
// ======================== TIME STEP ==========================
; L81
LOAD      F00099
MOV       D010210[Z013] D010250
; L82
LOAD      F00099
MAX       D010210 D010252 32
// ======================== ORIGIN ==========================
; L84
LOAD      M11094	// T)L_3rd MAND ORIGIN
AND NOT   M11080	// L_3rd MAND CYCLE RUN
OR        M01521	// L_P&P Y POWER ON
OR        M0002F	// INITIAL PLS
OR        M19102	// T)LEFT INITIAL
OUTP      M11096	// T)L_3rd MAND ORIGIN PLS
; L88
LOAD      M11096	// T)L_3rd MAND ORIGIN PLS
AND NOT   M1109A	// L_3rd MAND ORIGIN KP
LOAD NOT  M11096	// T)L_3rd MAND ORIGIN PLS
AND       M1109A	// L_3rd MAND ORIGIN KP
OR LOAD
AND NOT   M11080	// L_3rd MAND CYCLE RUN
AND NOT   M11078	// L_3rd MAND STEP INITIAL OK
AND       M01232	// LF ¢¬¨­AI ¨úE¢Ò¡À ¨ú¨¡¢¥O
OUT       M1109A	// L_3rd MAND ORIGIN KP
; L90
LOAD      M1109A	// L_3rd MAND ORIGIN KP
AND       F00093
OR        M11078	// L_3rd MAND STEP INITIAL OK
OUT       M1109B	// L_3rd MAND ORIGIN LAMP
; L92
LOAD NOT  M04070	// -
OR        M11060	// L_3rd BD Z ORIGIN->
AND       T0707	// -
AND       M1109A	// L_3rd MAND ORIGIN KP
AND NOT   M01571	// -
AND NOT   M03070	// -
AND       P00025	// L_1st ROTATE MANDREL BACKWARD
AND       T1110	// L_4th FPCB SUPPORT UP
OUT       M11060	// L_3rd BD Z ORIGIN->
; L94
LOAD NOT  M04060	// -
OR        M11061	// L_3rd ROT Y ORIGIN->
AND       T0706	// L_3rd SPK Y READY 2s
AND       M1109A	// L_3rd MAND ORIGIN KP
AND NOT   M01561	// L_3rd SPK Y POWER ON
AND NOT   M03060	// -
AND       P0004A	// -
AND       T1110	// L_4th FPCB SUPPORT UP
OUT       M11061	// L_3rd ROT Y ORIGIN->

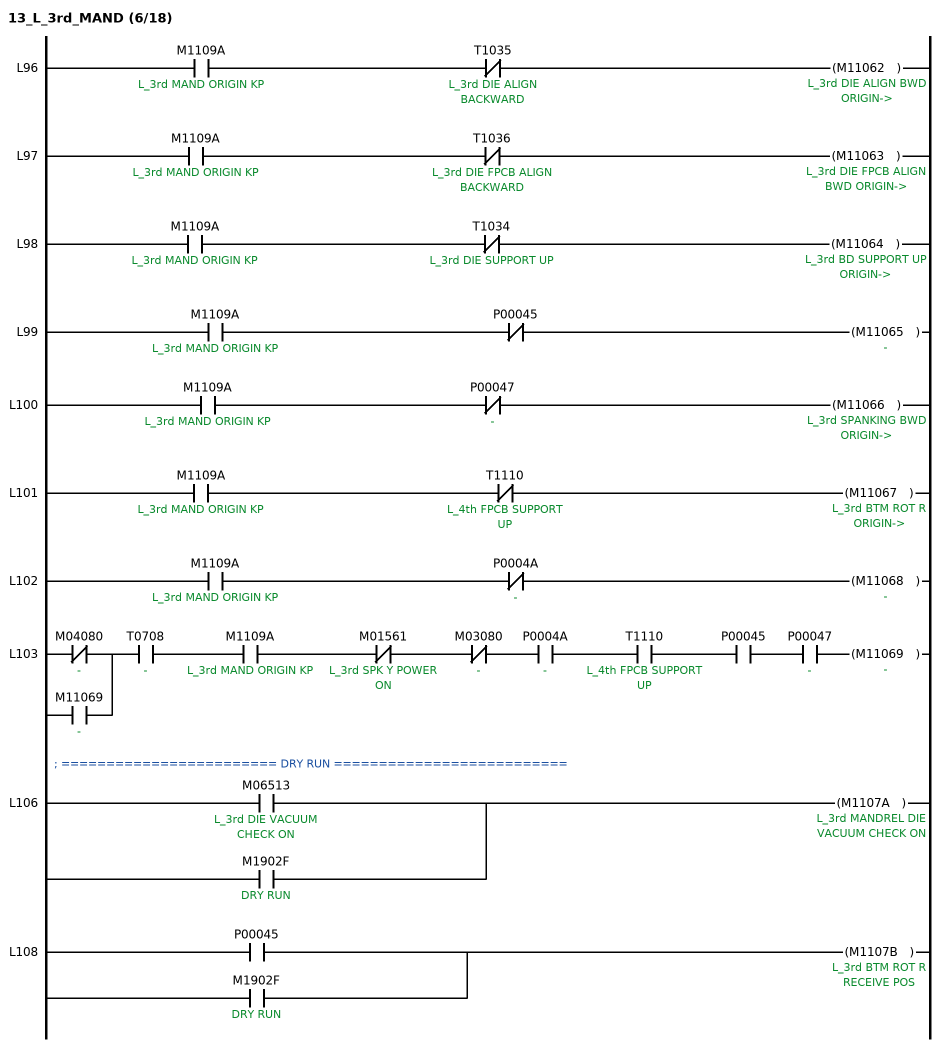
; L96
LOAD      M1109A	// L_3rd MAND ORIGIN KP
AND NOT   T1035	// L_3rd DIE ALIGN BACKWARD
OUT       M11062	// L_3rd DIE ALIGN BWD ORIGIN->
; L97
LOAD      M1109A	// L_3rd MAND ORIGIN KP
AND NOT   T1036	// L_3rd DIE FPCB ALIGN BACKWARD
OUT       M11063	// L_3rd DIE FPCB ALIGN BWD ORIGIN->
; L98
LOAD      M1109A	// L_3rd MAND ORIGIN KP
AND NOT   T1034	// L_3rd DIE SUPPORT UP
OUT       M11064	// L_3rd BD SUPPORT UP ORIGIN->
; L99
LOAD      M1109A	// L_3rd MAND ORIGIN KP
AND NOT   P00045
OUT       M11065	// -
; L100
LOAD      M1109A	// L_3rd MAND ORIGIN KP
AND NOT   P00047	// -
OUT       M11066	// L_3rd SPANKING BWD ORIGIN->
; L101
LOAD      M1109A	// L_3rd MAND ORIGIN KP
AND NOT   T1110	// L_4th FPCB SUPPORT UP
OUT       M11067	// L_3rd BTM ROT R ORIGIN->
; L102
LOAD      M1109A	// L_3rd MAND ORIGIN KP
AND NOT   P0004A	// -
OUT       M11068	// -
; L103
LOAD NOT  M04080	// -
OR        M11069	// -
AND       T0708	// -
AND       M1109A	// L_3rd MAND ORIGIN KP
AND NOT   M01561	// L_3rd SPK Y POWER ON
AND NOT   M03080	// -
AND       P0004A	// -
AND       T1110	// L_4th FPCB SUPPORT UP
AND       P00045
AND       P00047	// -
OUT       M11069	// -
// ======================== DRY RUN ==========================
; L106
LOAD      M06513	// L_3rd DIE VACUUM CHECK ON
OR        M1902F	// DRY RUN
OUT       M1107A	// L_3rd MANDREL DIE VACUUM CHECK ON
; L108
LOAD      P00045
OR        M1902F	// DRY RUN
OUT       M1107B	// L_3rd BTM ROT R RECEIVE POS

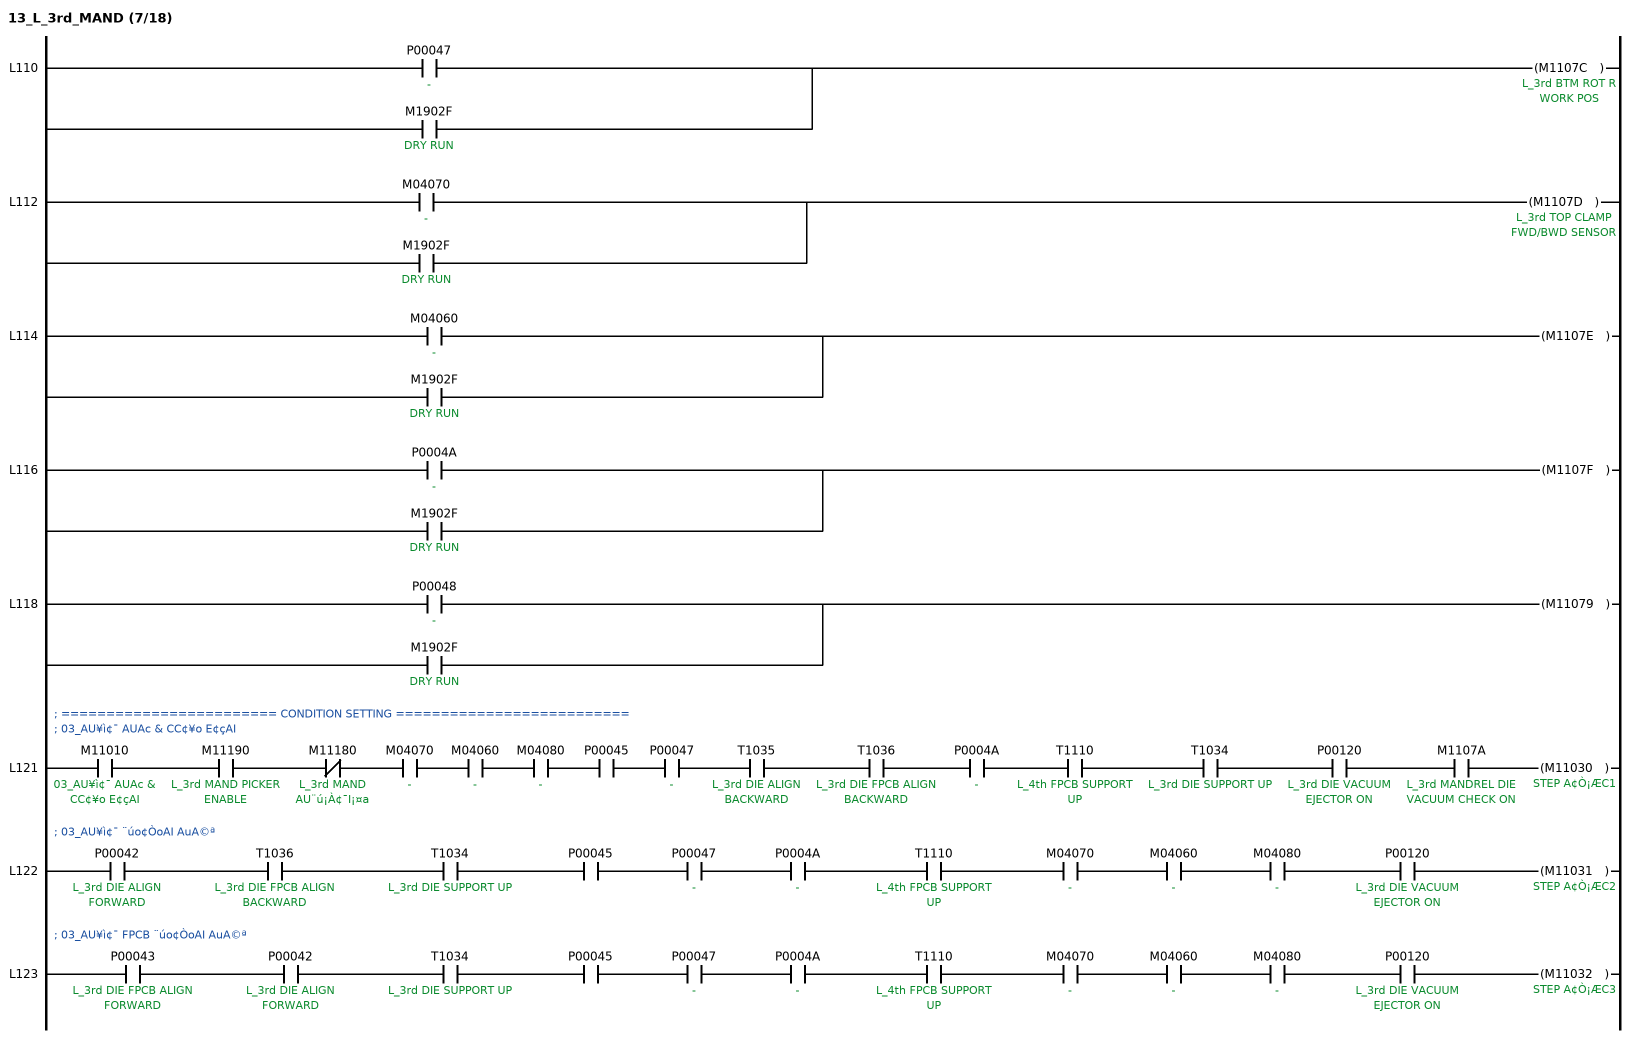
; L110
LOAD      P00047	// -
OR        M1902F	// DRY RUN
OUT       M1107C	// L_3rd BTM ROT R WORK POS
; L112
LOAD      M04070	// -
OR        M1902F	// DRY RUN
OUT       M1107D	// L_3rd TOP CLAMP FWD/BWD SENSOR
; L114
LOAD      M04060	// -
OR        M1902F	// DRY RUN
OUT       M1107E
; L116
LOAD      P0004A	// -
OR        M1902F	// DRY RUN
OUT       M1107F
; L118
LOAD      P00048	// -
OR        M1902F	// DRY RUN
OUT       M11079
// ======================== CONDITION SETTING ==========================
; L121
LOAD      M11010	// 03_AU¥ì¢¯ AUAc & CC¢¥o E¢çAI
AND       M11190	// L_3rd MAND PICKER ENABLE
AND NOT   M11180	// L_3rd MAND AU¨ú¡À¢¯I¡¤a
AND       M04070	// -
AND       M04060	// -
AND       M04080	// -
AND       P00045
AND       P00047	// -
AND       T1035	// L_3rd DIE ALIGN BACKWARD
AND       T1036	// L_3rd DIE FPCB ALIGN BACKWARD
AND       P0004A	// -
AND       T1110	// L_4th FPCB SUPPORT UP
AND       T1034	// L_3rd DIE SUPPORT UP
AND       P00120	// L_3rd DIE VACUUM EJECTOR ON
AND       M1107A	// L_3rd MANDREL DIE VACUUM CHECK ON
OUT       M11030	// STEP A¢Ò¡ÆC1
// output comment: 03_AU¥ì¢¯ AUAc & CC¢¥o E¢çAI
; L122
LOAD      P00042	// L_3rd DIE ALIGN FORWARD
AND       T1036	// L_3rd DIE FPCB ALIGN BACKWARD
AND       T1034	// L_3rd DIE SUPPORT UP
AND       P00045
AND       P00047	// -
AND       P0004A	// -
AND       T1110	// L_4th FPCB SUPPORT UP
AND       M04070	// -
AND       M04060	// -
AND       M04080	// -
AND       P00120	// L_3rd DIE VACUUM EJECTOR ON
OUT       M11031	// STEP A¢Ò¡ÆC2
// output comment: 03_AU¥ì¢¯ ¨úo¢ÒoAI AuA©ª
; L123
LOAD      P00043	// L_3rd DIE FPCB ALIGN FORWARD
AND       P00042	// L_3rd DIE ALIGN FORWARD
AND       T1034	// L_3rd DIE SUPPORT UP
AND       P00045
AND       P00047	// -
AND       P0004A	// -
AND       T1110	// L_4th FPCB SUPPORT UP
AND       M04070	// -
AND       M04060	// -
AND       M04080	// -
AND       P00120	// L_3rd DIE VACUUM EJECTOR ON
OUT       M11032	// STEP A¢Ò¡ÆC3
// output comment: 03_AU¥ì¢¯ FPCB ¨úo¢ÒoAI AuA©ª

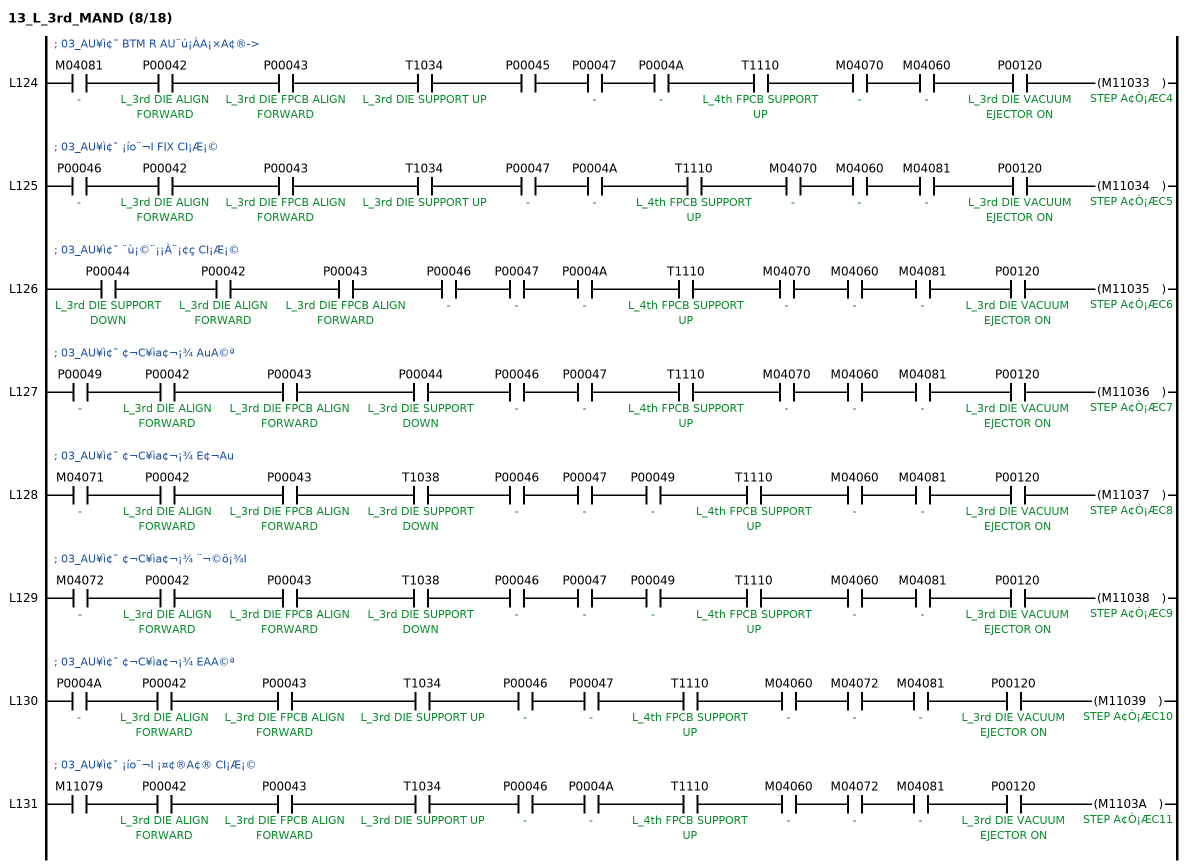
; L124
LOAD      M04081	// -
AND       P00042	// L_3rd DIE ALIGN FORWARD
AND       P00043	// L_3rd DIE FPCB ALIGN FORWARD
AND       T1034	// L_3rd DIE SUPPORT UP
AND       P00045
AND       P00047	// -
AND       P0004A	// -
AND       T1110	// L_4th FPCB SUPPORT UP
AND       M04070	// -
AND       M04060	// -
AND       P00120	// L_3rd DIE VACUUM EJECTOR ON
OUT       M11033	// STEP A¢Ò¡ÆC4
// output comment: 03_AU¥ì¢¯ BTM R AU¨ú¡ÀA¡×A¢®->
; L125
LOAD      P00046	// -
AND       P00042	// L_3rd DIE ALIGN FORWARD
AND       P00043	// L_3rd DIE FPCB ALIGN FORWARD
AND       T1034	// L_3rd DIE SUPPORT UP
AND       P00047	// -
AND       P0004A	// -
AND       T1110	// L_4th FPCB SUPPORT UP
AND       M04070	// -
AND       M04060	// -
AND       M04081	// -
AND       P00120	// L_3rd DIE VACUUM EJECTOR ON
OUT       M11034	// STEP A¢Ò¡ÆC5
// output comment: 03_AU¥ì¢¯ ¡ío¨¬I FIX CI¡Æ¡©
; L126
LOAD      P00044	// L_3rd DIE SUPPORT DOWN
AND       P00042	// L_3rd DIE ALIGN FORWARD
AND       P00043	// L_3rd DIE FPCB ALIGN FORWARD
AND       P00046	// -
AND       P00047	// -
AND       P0004A	// -
AND       T1110	// L_4th FPCB SUPPORT UP
AND       M04070	// -
AND       M04060	// -
AND       M04081	// -
AND       P00120	// L_3rd DIE VACUUM EJECTOR ON
OUT       M11035	// STEP A¢Ò¡ÆC6
// output comment: 03_AU¥ì¢¯ ¨ù¡©¨¡¡À¨¡¢ç CI¡Æ¡©
; L127
LOAD      P00049	// -
AND       P00042	// L_3rd DIE ALIGN FORWARD
AND       P00043	// L_3rd DIE FPCB ALIGN FORWARD
AND       P00044	// L_3rd DIE SUPPORT DOWN
AND       P00046	// -
AND       P00047	// -
AND       T1110	// L_4th FPCB SUPPORT UP
AND       M04070	// -
AND       M04060	// -
AND       M04081	// -
AND       P00120	// L_3rd DIE VACUUM EJECTOR ON
OUT       M11036	// STEP A¢Ò¡ÆC7
// output comment: 03_AU¥ì¢¯ ¢¬C¥ìa¢¬¡¾ AuA©ª
; L128
LOAD      M04071	// -
AND       P00042	// L_3rd DIE ALIGN FORWARD
AND       P00043	// L_3rd DIE FPCB ALIGN FORWARD
AND       T1038	// L_3rd DIE SUPPORT DOWN
AND       P00046	// -
AND       P00047	// -
AND       P00049	// -
AND       T1110	// L_4th FPCB SUPPORT UP
AND       M04060	// -
AND       M04081	// -
AND       P00120	// L_3rd DIE VACUUM EJECTOR ON
OUT       M11037	// STEP A¢Ò¡ÆC8
// output comment: 03_AU¥ì¢¯ ¢¬C¥ìa¢¬¡¾ E¢¬Au
; L129
LOAD      M04072	// -
AND       P00042	// L_3rd DIE ALIGN FORWARD
AND       P00043	// L_3rd DIE FPCB ALIGN FORWARD
AND       T1038	// L_3rd DIE SUPPORT DOWN
AND       P00046	// -
AND       P00047	// -
AND       P00049	// -
AND       T1110	// L_4th FPCB SUPPORT UP
AND       M04060	// -
AND       M04081	// -
AND       P00120	// L_3rd DIE VACUUM EJECTOR ON
OUT       M11038	// STEP A¢Ò¡ÆC9
// output comment: 03_AU¥ì¢¯ ¢¬C¥ìa¢¬¡¾ ¨¬©ö¡¾I
; L130
LOAD      P0004A	// -
AND       P00042	// L_3rd DIE ALIGN FORWARD
AND       P00043	// L_3rd DIE FPCB ALIGN FORWARD
AND       T1034	// L_3rd DIE SUPPORT UP
AND       P00046	// -
AND       P00047	// -
AND       T1110	// L_4th FPCB SUPPORT UP
AND       M04060	// -
AND       M04072	// -
AND       M04081	// -
AND       P00120	// L_3rd DIE VACUUM EJECTOR ON
OUT       M11039	// STEP A¢Ò¡ÆC10
// output comment: 03_AU¥ì¢¯ ¢¬C¥ìa¢¬¡¾ EAA©ª
; L131
LOAD      M11079
AND       P00042	// L_3rd DIE ALIGN FORWARD
AND       P00043	// L_3rd DIE FPCB ALIGN FORWARD
AND       T1034	// L_3rd DIE SUPPORT UP
AND       P00046	// -
AND       P0004A	// -
AND       T1110	// L_4th FPCB SUPPORT UP
AND       M04060	// -
AND       M04072	// -
AND       M04081	// -
AND       P00120	// L_3rd DIE VACUUM EJECTOR ON
OUT       M1103A	// STEP A¢Ò¡ÆC11
// output comment: 03_AU¥ì¢¯ ¡ío¨¬I ¡¤¢®A¢® CI¡Æ¡©

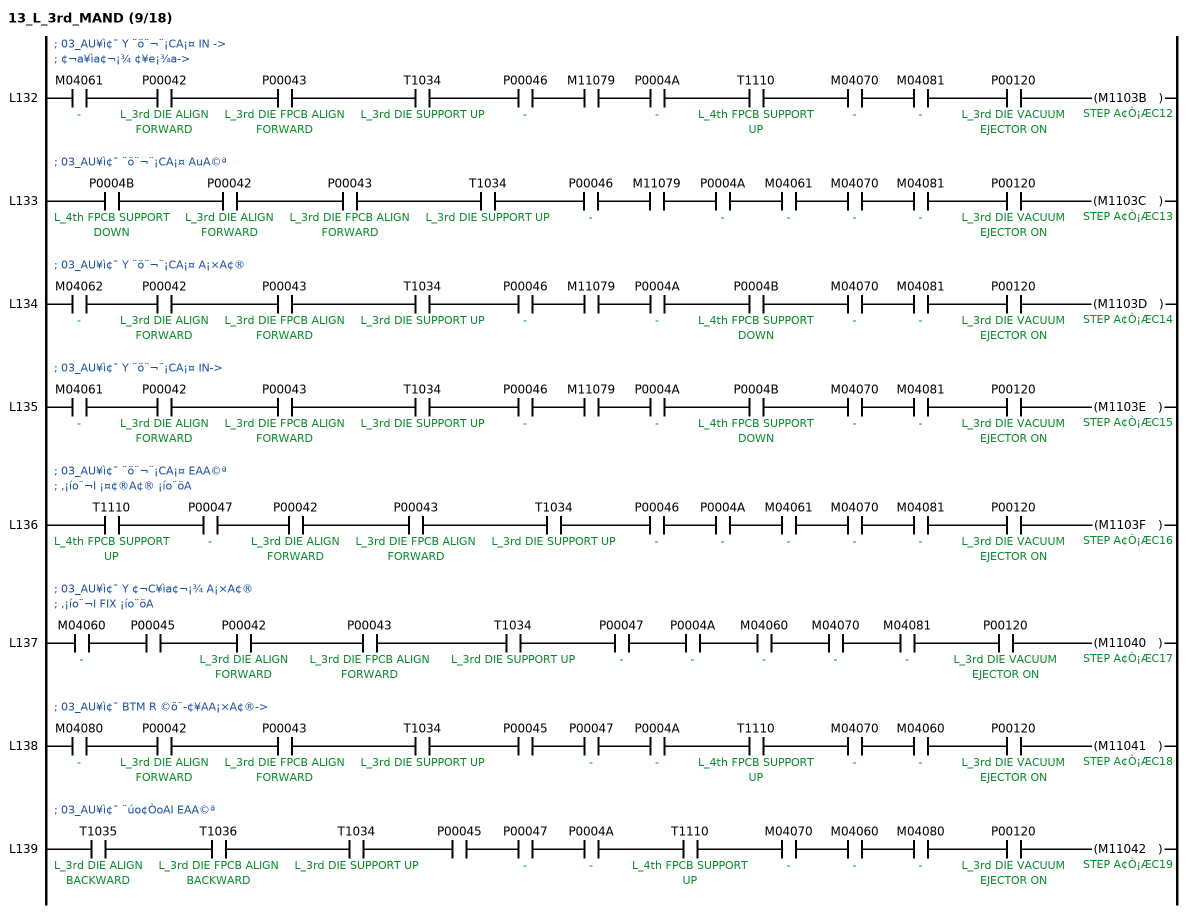
; L132
LOAD      M04061	// -
AND       P00042	// L_3rd DIE ALIGN FORWARD
AND       P00043	// L_3rd DIE FPCB ALIGN FORWARD
AND       T1034	// L_3rd DIE SUPPORT UP
AND       P00046	// -
AND       M11079
AND       P0004A	// -
AND       T1110	// L_4th FPCB SUPPORT UP
AND       M04070	// -
AND       M04081	// -
AND       P00120	// L_3rd DIE VACUUM EJECTOR ON
OUT       M1103B	// STEP A¢Ò¡ÆC12
// output comment: 03_AU¥ì¢¯ Y ¨ö¨¬¨¡CA¡¤ IN -> ¢¬a¥ìa¢¬¡¾ ¢¥e¡¾a->
; L133
LOAD      P0004B	// L_4th FPCB SUPPORT DOWN
AND       P00042	// L_3rd DIE ALIGN FORWARD
AND       P00043	// L_3rd DIE FPCB ALIGN FORWARD
AND       T1034	// L_3rd DIE SUPPORT UP
AND       P00046	// -
AND       M11079
AND       P0004A	// -
AND       M04061	// -
AND       M04070	// -
AND       M04081	// -
AND       P00120	// L_3rd DIE VACUUM EJECTOR ON
OUT       M1103C	// STEP A¢Ò¡ÆC13
// output comment: 03_AU¥ì¢¯ ¨ö¨¬¨¡CA¡¤ AuA©ª
; L134
LOAD      M04062	// -
AND       P00042	// L_3rd DIE ALIGN FORWARD
AND       P00043	// L_3rd DIE FPCB ALIGN FORWARD
AND       T1034	// L_3rd DIE SUPPORT UP
AND       P00046	// -
AND       M11079
AND       P0004A	// -
AND       P0004B	// L_4th FPCB SUPPORT DOWN
AND       M04070	// -
AND       M04081	// -
AND       P00120	// L_3rd DIE VACUUM EJECTOR ON
OUT       M1103D	// STEP A¢Ò¡ÆC14
// output comment: 03_AU¥ì¢¯ Y ¨ö¨¬¨¡CA¡¤ A¡×A¢®
; L135
LOAD      M04061	// -
AND       P00042	// L_3rd DIE ALIGN FORWARD
AND       P00043	// L_3rd DIE FPCB ALIGN FORWARD
AND       T1034	// L_3rd DIE SUPPORT UP
AND       P00046	// -
AND       M11079
AND       P0004A	// -
AND       P0004B	// L_4th FPCB SUPPORT DOWN
AND       M04070	// -
AND       M04081	// -
AND       P00120	// L_3rd DIE VACUUM EJECTOR ON
OUT       M1103E	// STEP A¢Ò¡ÆC15
// output comment: 03_AU¥ì¢¯ Y ¨ö¨¬¨¡CA¡¤ IN->
; L136
LOAD      T1110	// L_4th FPCB SUPPORT UP
AND       P00047	// -
AND       P00042	// L_3rd DIE ALIGN FORWARD
AND       P00043	// L_3rd DIE FPCB ALIGN FORWARD
AND       T1034	// L_3rd DIE SUPPORT UP
AND       P00046	// -
AND       P0004A	// -
AND       M04061	// -
AND       M04070	// -
AND       M04081	// -
AND       P00120	// L_3rd DIE VACUUM EJECTOR ON
OUT       M1103F	// STEP A¢Ò¡ÆC16
// output comment: 03_AU¥ì¢¯ ¨ö¨¬¨¡CA¡¤ EAA©ª ,¡ío¨¬I ¡¤¢®A¢® ¡ío¨öA
; L137
LOAD      M04060	// -
AND       P00045
AND       P00042	// L_3rd DIE ALIGN FORWARD
AND       P00043	// L_3rd DIE FPCB ALIGN FORWARD
AND       T1034	// L_3rd DIE SUPPORT UP
AND       P00047	// -
AND       P0004A	// -
AND       M04060	// -
AND       M04070	// -
AND       M04081	// -
AND       P00120	// L_3rd DIE VACUUM EJECTOR ON
OUT       M11040	// STEP A¢Ò¡ÆC17
// output comment: 03_AU¥ì¢¯ Y ¢¬C¥ìa¢¬¡¾ A¡×A¢® ,¡ío¨¬I FIX ¡ío¨öA
; L138
LOAD      M04080	// -
AND       P00042	// L_3rd DIE ALIGN FORWARD
AND       P00043	// L_3rd DIE FPCB ALIGN FORWARD
AND       T1034	// L_3rd DIE SUPPORT UP
AND       P00045
AND       P00047	// -
AND       P0004A	// -
AND       T1110	// L_4th FPCB SUPPORT UP
AND       M04070	// -
AND       M04060	// -
AND       P00120	// L_3rd DIE VACUUM EJECTOR ON
OUT       M11041	// STEP A¢Ò¡ÆC18
// output comment: 03_AU¥ì¢¯ BTM R ©ö¨­¢¥AA¡×A¢®->
; L139
LOAD      T1035	// L_3rd DIE ALIGN BACKWARD
AND       T1036	// L_3rd DIE FPCB ALIGN BACKWARD
AND       T1034	// L_3rd DIE SUPPORT UP
AND       P00045
AND       P00047	// -
AND       P0004A	// -
AND       T1110	// L_4th FPCB SUPPORT UP
AND       M04070	// -
AND       M04060	// -
AND       M04080	// -
AND       P00120	// L_3rd DIE VACUUM EJECTOR ON
OUT       M11042	// STEP A¢Ò¡ÆC19
// output comment: 03_AU¥ì¢¯ ¨úo¢ÒoAI EAA©ª

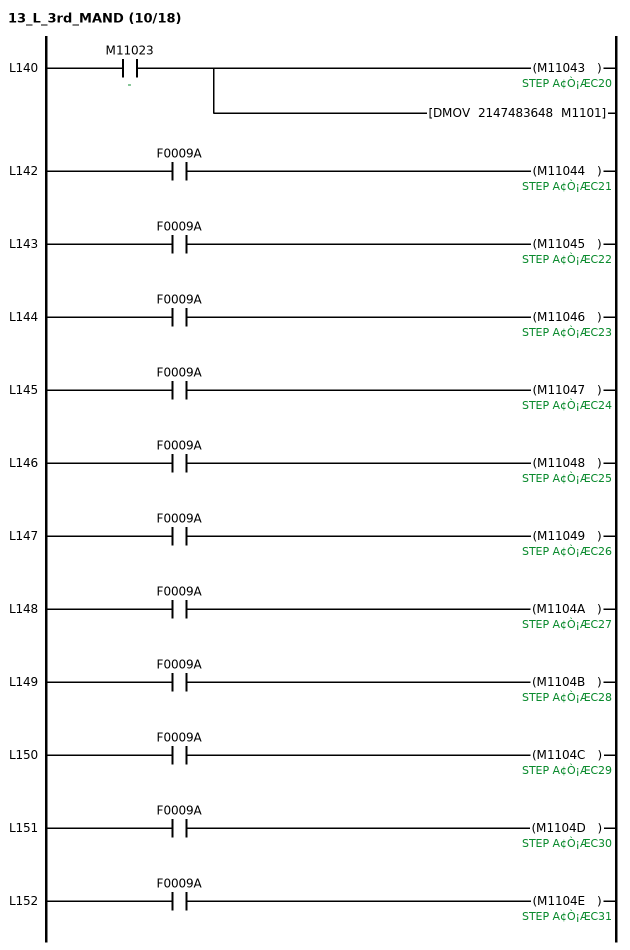
; L140
LOAD      M11023	// -
OUT       M11043	// STEP A¢Ò¡ÆC20
DMOV      2147483648 M1101
; L142
LOAD      F0009A
OUT       M11044	// STEP A¢Ò¡ÆC21
; L143
LOAD      F0009A
OUT       M11045	// STEP A¢Ò¡ÆC22
; L144
LOAD      F0009A
OUT       M11046	// STEP A¢Ò¡ÆC23
; L145
LOAD      F0009A
OUT       M11047	// STEP A¢Ò¡ÆC24
; L146
LOAD      F0009A
OUT       M11048	// STEP A¢Ò¡ÆC25
; L147
LOAD      F0009A
OUT       M11049	// STEP A¢Ò¡ÆC26
; L148
LOAD      F0009A
OUT       M1104A	// STEP A¢Ò¡ÆC27
; L149
LOAD      F0009A
OUT       M1104B	// STEP A¢Ò¡ÆC28
; L150
LOAD      F0009A
OUT       M1104C	// STEP A¢Ò¡ÆC29
; L151
LOAD      F0009A
OUT       M1104D	// STEP A¢Ò¡ÆC30
; L152
LOAD      F0009A
OUT       M1104E	// STEP A¢Ò¡ÆC31

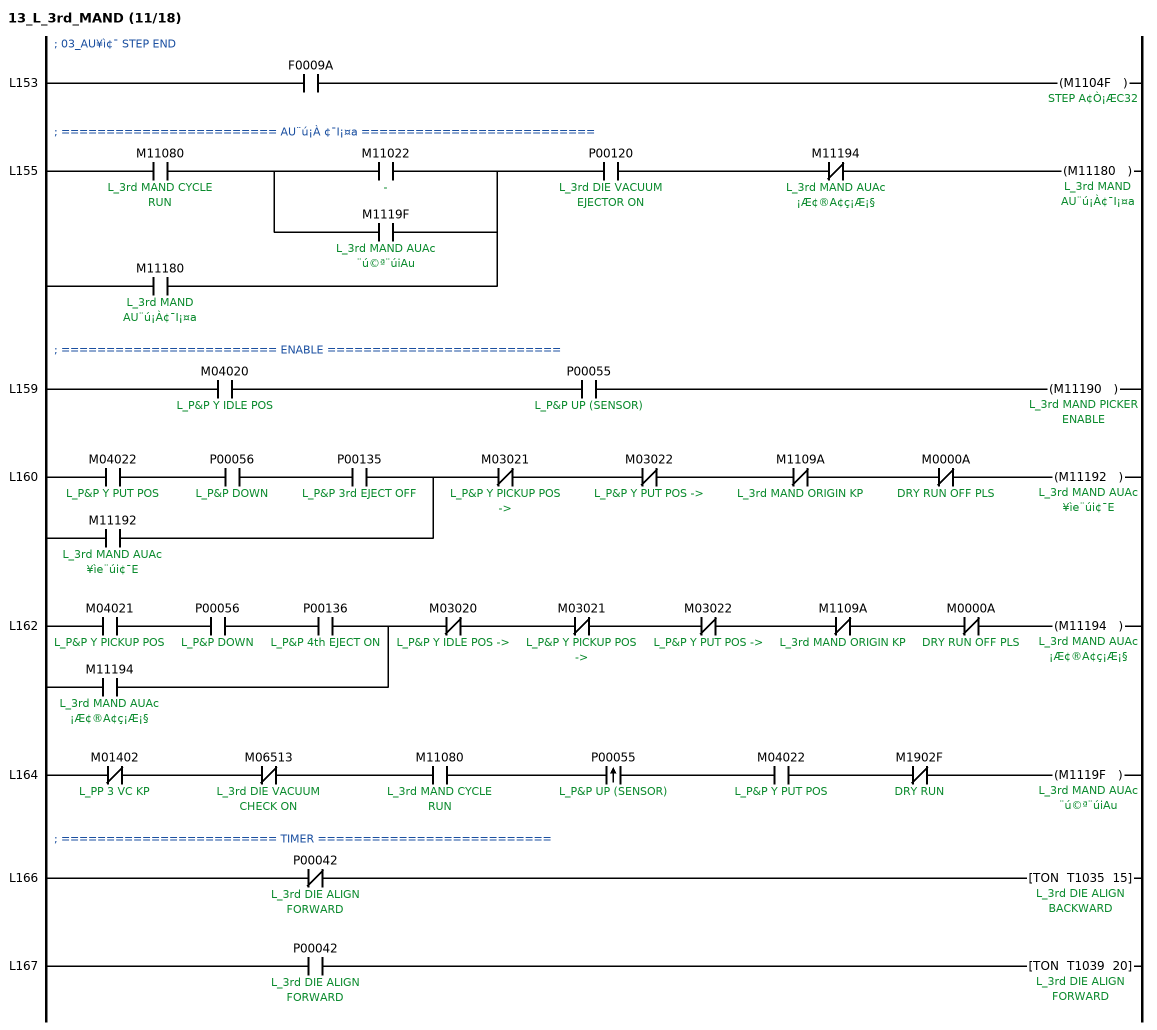
; L153
LOAD      F0009A
OUT       M1104F	// STEP A¢Ò¡ÆC32
// output comment: 03_AU¥ì¢¯ STEP END
// ======================== AU¨ú¡À ¢¯I¡¤a ==========================
; L155
LOAD      M11080	// L_3rd MAND CYCLE RUN
LOAD      M11022	// -
OR        M1119F	// L_3rd MAND AUAc ¨ú©ª¨úiAu
AND LOAD
OR        M11180	// L_3rd MAND AU¨ú¡À¢¯I¡¤a
AND       P00120	// L_3rd DIE VACUUM EJECTOR ON
AND NOT   M11194	// L_3rd MAND AUAc ¡Æ¢®A¢ç¡Æ¡§
OUT       M11180	// L_3rd MAND AU¨ú¡À¢¯I¡¤a
// ======================== ENABLE ==========================
; L159
LOAD      M04020	// L_P&P Y IDLE POS
AND       P00055	// L_P&P UP (SENSOR)
OUT       M11190	// L_3rd MAND PICKER ENABLE
; L160
LOAD      M04022	// L_P&P Y PUT POS
AND       P00056	// L_P&P DOWN
AND       P00135	// L_P&P 3rd EJECT OFF
OR        M11192	// L_3rd MAND AUAc ¥ìe¨úi¢¯E
AND NOT   M03021	// L_P&P Y PICKUP POS ->
AND NOT   M03022	// L_P&P Y PUT POS ->
AND NOT   M1109A	// L_3rd MAND ORIGIN KP
AND NOT   M0000A	// DRY RUN OFF PLS
OUT       M11192	// L_3rd MAND AUAc ¥ìe¨úi¢¯E
; L162
LOAD      M04021	// L_P&P Y PICKUP POS
AND       P00056	// L_P&P DOWN
AND       P00136	// L_P&P 4th EJECT ON
OR        M11194	// L_3rd MAND AUAc ¡Æ¢®A¢ç¡Æ¡§
AND NOT   M03020	// L_P&P Y IDLE POS ->
AND NOT   M03021	// L_P&P Y PICKUP POS ->
AND NOT   M03022	// L_P&P Y PUT POS ->
AND NOT   M1109A	// L_3rd MAND ORIGIN KP
AND NOT   M0000A	// DRY RUN OFF PLS
OUT       M11194	// L_3rd MAND AUAc ¡Æ¢®A¢ç¡Æ¡§
; L164
LOAD NOT  M01402	// L_PP 3 VC KP
AND NOT   M06513	// L_3rd DIE VACUUM CHECK ON
AND       M11080	// L_3rd MAND CYCLE RUN
ANDP      P00055	// L_P&P UP (SENSOR)
AND       M04022	// L_P&P Y PUT POS
AND NOT   M1902F	// DRY RUN
OUT       M1119F	// L_3rd MAND AUAc ¨ú©ª¨úiAu
// ======================== TIMER ==========================
; L166
LOAD NOT  P00042	// L_3rd DIE ALIGN FORWARD
TON       T1035 15	// L_3rd DIE ALIGN BACKWARD
; L167
LOAD      P00042	// L_3rd DIE ALIGN FORWARD
TON       T1039 20	// L_3rd DIE ALIGN FORWARD

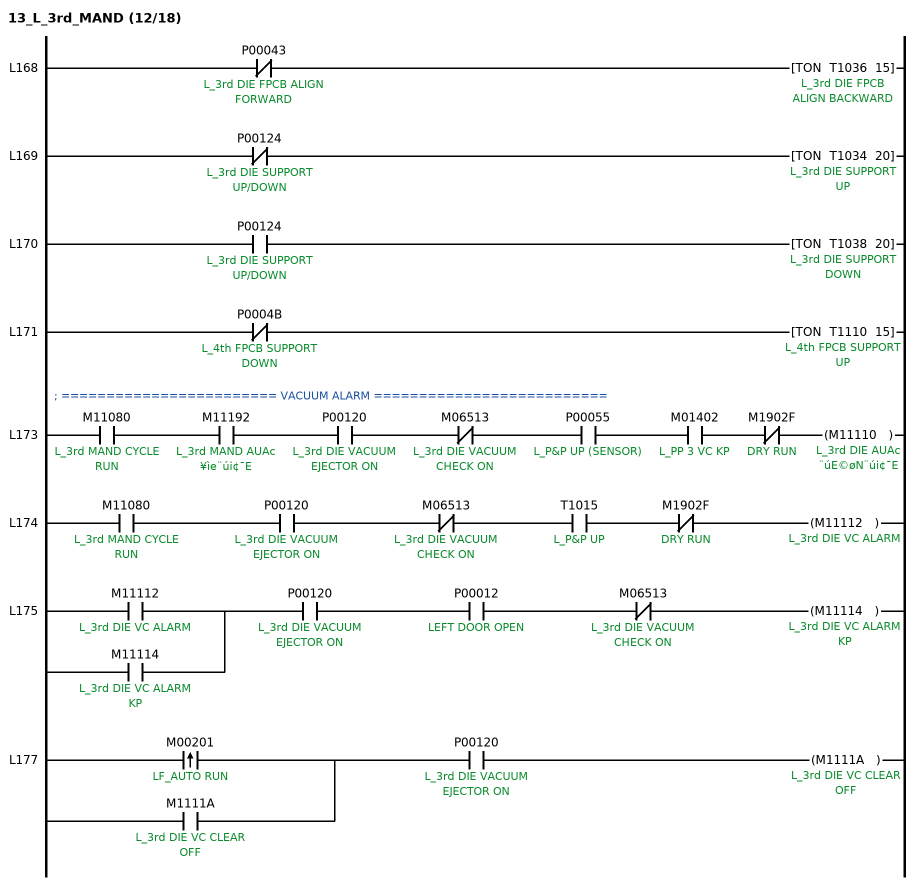
; L168
LOAD NOT  P00043	// L_3rd DIE FPCB ALIGN FORWARD
TON       T1036 15	// L_3rd DIE FPCB ALIGN BACKWARD
; L169
LOAD NOT  P00124	// L_3rd DIE SUPPORT UP/DOWN
TON       T1034 20	// L_3rd DIE SUPPORT UP
; L170
LOAD      P00124	// L_3rd DIE SUPPORT UP/DOWN
TON       T1038 20	// L_3rd DIE SUPPORT DOWN
; L171
LOAD NOT  P0004B	// L_4th FPCB SUPPORT DOWN
TON       T1110 15	// L_4th FPCB SUPPORT UP
// ======================== VACUUM ALARM ==========================
; L173
LOAD      M11080	// L_3rd MAND CYCLE RUN
AND       M11192	// L_3rd MAND AUAc ¥ìe¨úi¢¯E
AND       P00120	// L_3rd DIE VACUUM EJECTOR ON
AND NOT   M06513	// L_3rd DIE VACUUM CHECK ON
AND       P00055	// L_P&P UP (SENSOR)
AND       M01402	// L_PP 3 VC KP
AND NOT   M1902F	// DRY RUN
OUT       M11110	// L_3rd DIE AUAc ¨úE©øN¨úi¢¯E
; L174
LOAD      M11080	// L_3rd MAND CYCLE RUN
AND       P00120	// L_3rd DIE VACUUM EJECTOR ON
AND NOT   M06513	// L_3rd DIE VACUUM CHECK ON
AND       T1015	// L_P&P UP
AND NOT   M1902F	// DRY RUN
OUT       M11112	// L_3rd DIE VC ALARM
; L175
LOAD      M11112	// L_3rd DIE VC ALARM
OR        M11114	// L_3rd DIE VC ALARM KP
AND       P00120	// L_3rd DIE VACUUM EJECTOR ON
AND       P00012	// LEFT DOOR OPEN
AND NOT   M06513	// L_3rd DIE VACUUM CHECK ON
OUT       M11114	// L_3rd DIE VC ALARM KP
; L177
LOADP     M00201	// LF_AUTO RUN
OR        M1111A	// L_3rd DIE VC CLEAR OFF
AND       P00120	// L_3rd DIE VACUUM EJECTOR ON
OUT       M1111A	// L_3rd DIE VC CLEAR OFF

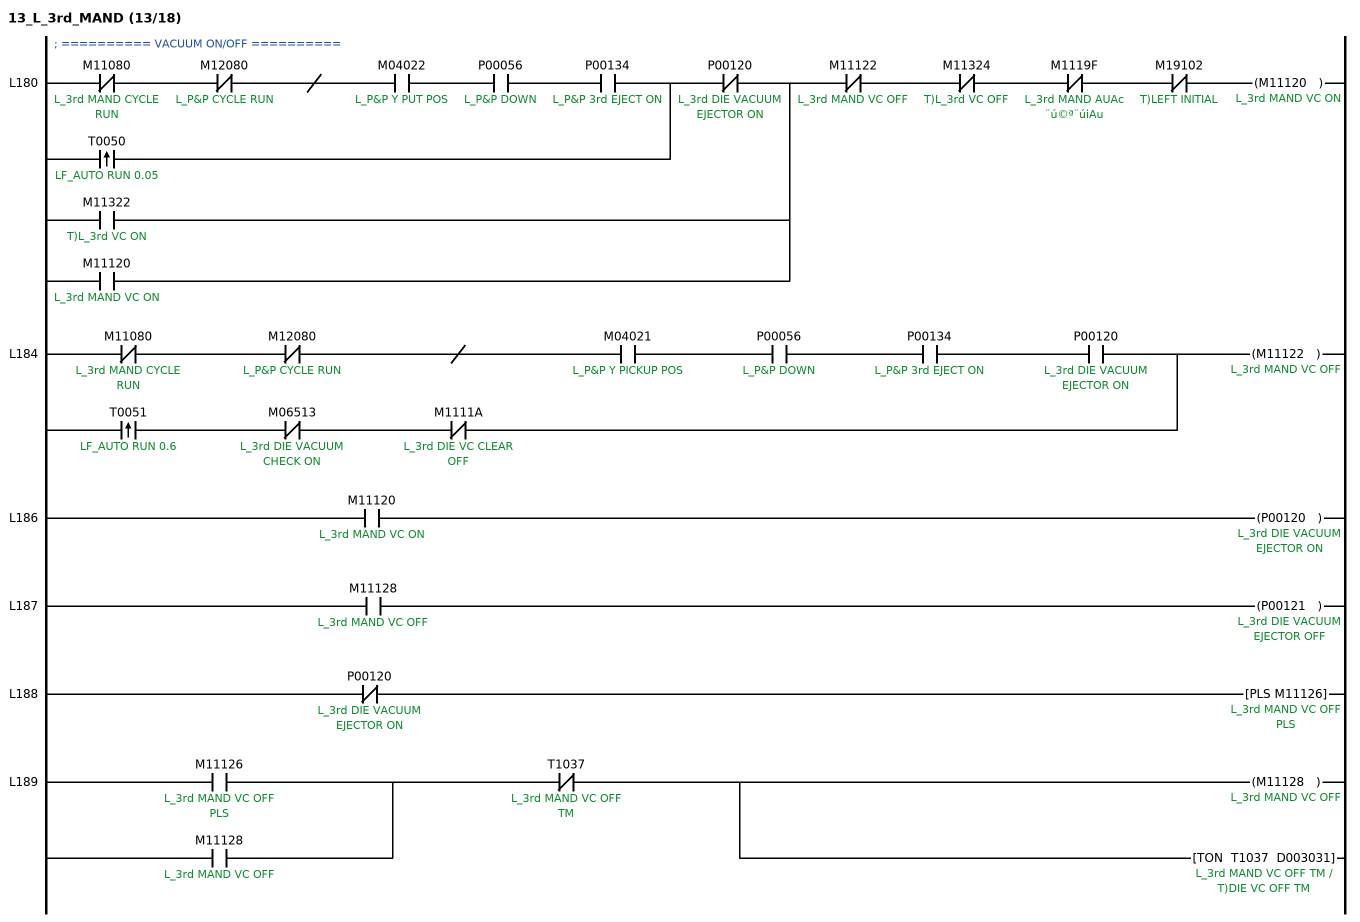
// ========== VACUUM ON/OFF ==========
; L180
LOAD NOT  M11080	// L_3rd MAND CYCLE RUN
AND NOT   M12080	// L_P&P CYCLE RUN
NOT
AND       M04022	// L_P&P Y PUT POS
AND       P00056	// L_P&P DOWN
AND       P00134	// L_P&P 3rd EJECT ON
ORP       T0050	// LF_AUTO RUN 0.05
AND NOT   P00120	// L_3rd DIE VACUUM EJECTOR ON
OR        M11322	// T)L_3rd VC ON
OR        M11120	// L_3rd MAND VC ON
AND NOT   M11122	// L_3rd MAND VC OFF
AND NOT   M11324	// T)L_3rd VC OFF
AND NOT   M1119F	// L_3rd MAND AUAc ¨ú©ª¨úiAu
AND NOT   M19102	// T)LEFT INITIAL
OUT       M11120	// L_3rd MAND VC ON
; L184
LOAD NOT  M11080	// L_3rd MAND CYCLE RUN
AND NOT   M12080	// L_P&P CYCLE RUN
NOT
AND       M04021	// L_P&P Y PICKUP POS
AND       P00056	// L_P&P DOWN
AND       P00134	// L_P&P 3rd EJECT ON
AND       P00120	// L_3rd DIE VACUUM EJECTOR ON
LOADP     T0051	// LF_AUTO RUN 0.6
AND NOT   M06513	// L_3rd DIE VACUUM CHECK ON
AND NOT   M1111A	// L_3rd DIE VC CLEAR OFF
OR LOAD
OUT       M11122	// L_3rd MAND VC OFF
; L186
LOAD      M11120	// L_3rd MAND VC ON
OUT       P00120	// L_3rd DIE VACUUM EJECTOR ON
; L187
LOAD      M11128	// L_3rd MAND VC OFF
OUT       P00121	// L_3rd DIE VACUUM EJECTOR OFF
; L188
LOAD NOT  P00120	// L_3rd DIE VACUUM EJECTOR ON
OUTP      M11126	// L_3rd MAND VC OFF PLS
; L189
LOAD      M11126	// L_3rd MAND VC OFF PLS
OR        M11128	// L_3rd MAND VC OFF
AND NOT   T1037	// L_3rd MAND VC OFF TM
OUT       M11128	// L_3rd MAND VC OFF
TON       T1037 D003031	// L_3rd MAND VC OFF TM / T)DIE VC OFF TM

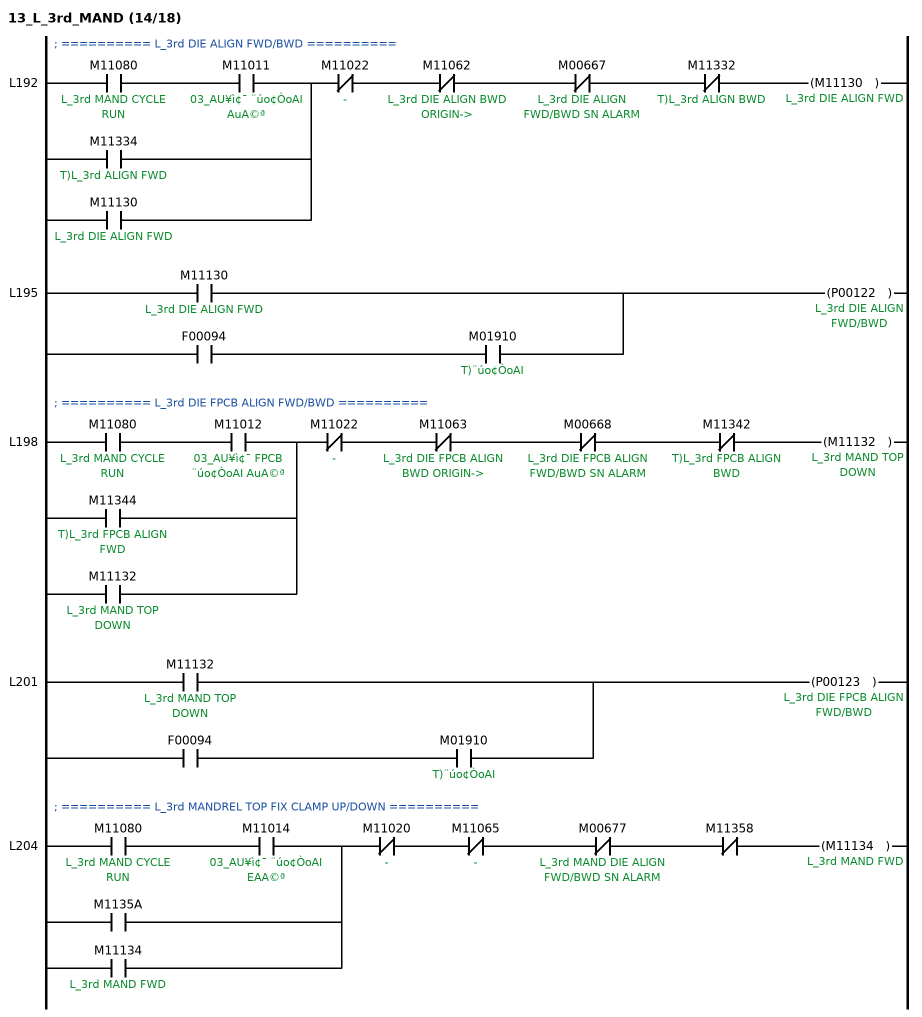
// ========== L_3rd DIE ALIGN FWD/BWD ==========
; L192
LOAD      M11080	// L_3rd MAND CYCLE RUN
AND       M11011	// 03_AU¥ì¢¯ ¨úo¢ÒoAI AuA©ª
OR        M11334	// T)L_3rd ALIGN FWD
OR        M11130	// L_3rd DIE ALIGN FWD
AND NOT   M11022	// -
AND NOT   M11062	// L_3rd DIE ALIGN BWD ORIGIN->
AND NOT   M00667	// L_3rd DIE ALIGN FWD/BWD SN ALARM
AND NOT   M11332	// T)L_3rd ALIGN BWD
OUT       M11130	// L_3rd DIE ALIGN FWD
; L195
LOAD      M11130	// L_3rd DIE ALIGN FWD
LOAD      F00094
AND       M01910	// T)¨úo¢ÒoAI
OR LOAD
OUT       P00122	// L_3rd DIE ALIGN FWD/BWD
// ========== L_3rd DIE FPCB ALIGN FWD/BWD ==========
; L198
LOAD      M11080	// L_3rd MAND CYCLE RUN
AND       M11012	// 03_AU¥ì¢¯ FPCB ¨úo¢ÒoAI AuA©ª
OR        M11344	// T)L_3rd FPCB ALIGN FWD
OR        M11132	// L_3rd MAND TOP DOWN
AND NOT   M11022	// -
AND NOT   M11063	// L_3rd DIE FPCB ALIGN BWD ORIGIN->
AND NOT   M00668	// L_3rd DIE FPCB ALIGN FWD/BWD SN ALARM
AND NOT   M11342	// T)L_3rd FPCB ALIGN BWD
OUT       M11132	// L_3rd MAND TOP DOWN
; L201
LOAD      M11132	// L_3rd MAND TOP DOWN
LOAD      F00094
AND       M01910	// T)¨úo¢ÒoAI
OR LOAD
OUT       P00123	// L_3rd DIE FPCB ALIGN FWD/BWD
// ========== L_3rd MANDREL TOP FIX CLAMP UP/DOWN ==========
; L204
LOAD      M11080	// L_3rd MAND CYCLE RUN
AND       M11014	// 03_AU¥ì¢¯ ¨úo¢ÒoAI EAA©ª
OR        M1135A
OR        M11134	// L_3rd MAND FWD
AND NOT   M11020	// -
AND NOT   M11065	// -
AND NOT   M00677	// L_3rd MAND DIE ALIGN FWD/BWD SN ALARM
AND NOT   M11358
OUT       M11134	// L_3rd MAND FWD

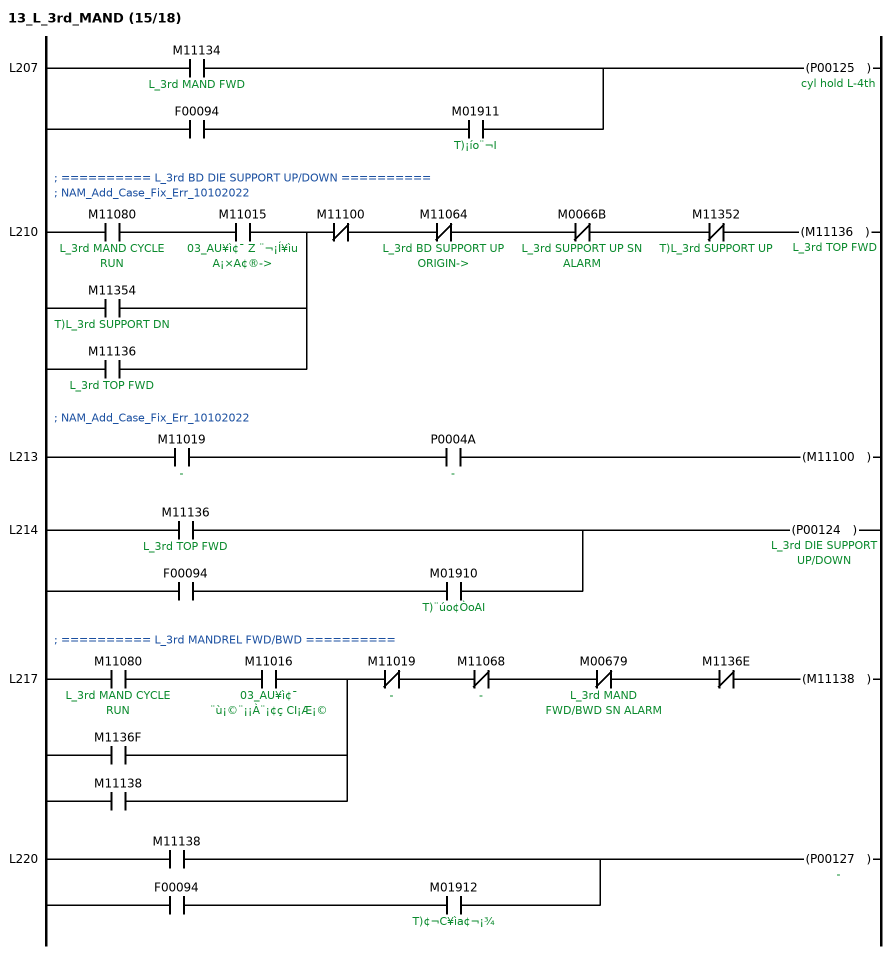
; L207
LOAD      M11134	// L_3rd MAND FWD
LOAD      F00094
AND       M01911	// T)¡ío¨¬I
OR LOAD
OUT       P00125	// cyl hold L-4th
// ========== L_3rd BD DIE SUPPORT UP/DOWN ==========
; L210
LOAD      M11080	// L_3rd MAND CYCLE RUN
AND       M11015	// 03_AU¥ì¢¯ Z ¨¬¡Í¥ìu A¡×A¢®->
OR        M11354	// T)L_3rd SUPPORT DN
OR        M11136	// L_3rd TOP FWD
AND NOT   M11100
AND NOT   M11064	// L_3rd BD SUPPORT UP ORIGIN->
AND NOT   M0066B	// L_3rd SUPPORT UP SN ALARM
AND NOT   M11352	// T)L_3rd SUPPORT UP
OUT       M11136	// L_3rd TOP FWD
// output comment: NAM_Add_Case_Fix_Err_10102022
; L213
LOAD      M11019	// -
AND       P0004A	// -
OUT       M11100
// output comment: NAM_Add_Case_Fix_Err_10102022
; L214
LOAD      M11136	// L_3rd TOP FWD
LOAD      F00094
AND       M01910	// T)¨úo¢ÒoAI
OR LOAD
OUT       P00124	// L_3rd DIE SUPPORT UP/DOWN
// ========== L_3rd MANDREL FWD/BWD ==========
; L217
LOAD      M11080	// L_3rd MAND CYCLE RUN
AND       M11016	// 03_AU¥ì¢¯ ¨ù¡©¨¡¡À¨¡¢ç CI¡Æ¡©
OR        M1136F
OR        M11138
AND NOT   M11019	// -
AND NOT   M11068	// -
AND NOT   M00679	// L_3rd MAND FWD/BWD SN ALARM
AND NOT   M1136E
OUT       M11138
; L220
LOAD      M11138
LOAD      F00094
AND       M01912	// T)¢¬C¥ìa¢¬¡¾
OR LOAD
OUT       P00127	// -

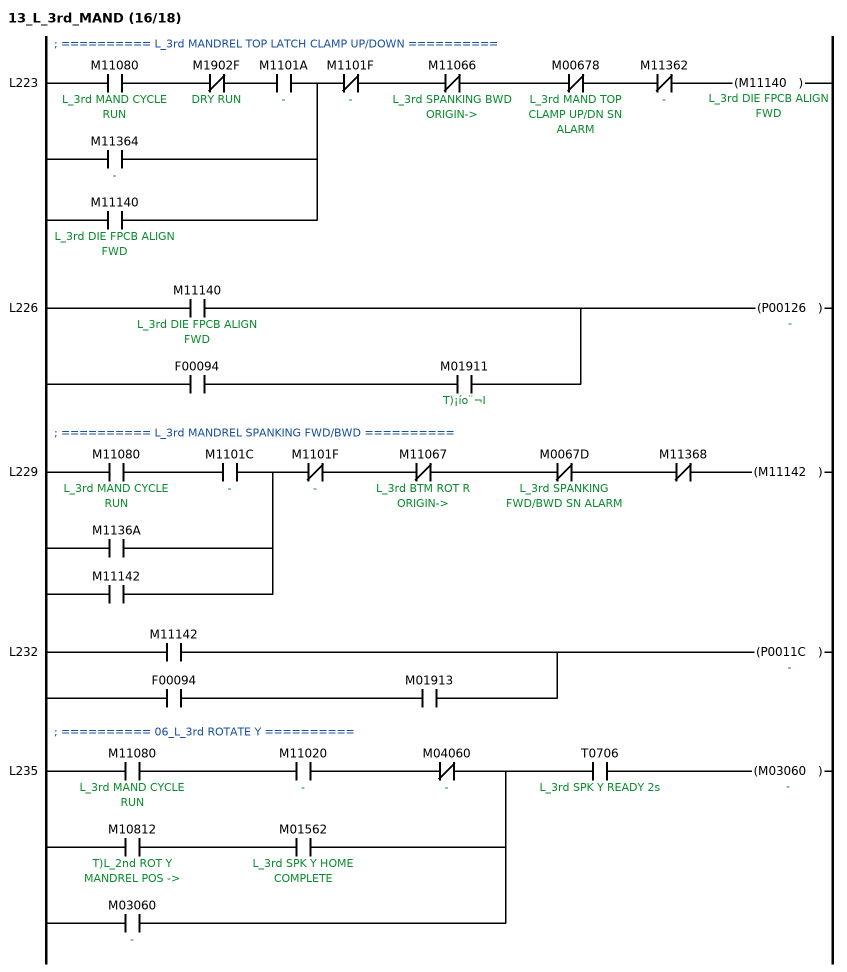
// ========== L_3rd MANDREL TOP LATCH CLAMP UP/DOWN ==========
; L223
LOAD      M11080	// L_3rd MAND CYCLE RUN
AND NOT   M1902F	// DRY RUN
AND       M1101A	// -
OR        M11364	// -
OR        M11140	// L_3rd DIE FPCB ALIGN FWD
AND NOT   M1101F	// -
AND NOT   M11066	// L_3rd SPANKING BWD ORIGIN->
AND NOT   M00678	// L_3rd MAND TOP CLAMP UP/DN SN ALARM
AND NOT   M11362	// -
OUT       M11140	// L_3rd DIE FPCB ALIGN FWD
; L226
LOAD      M11140	// L_3rd DIE FPCB ALIGN FWD
LOAD      F00094
AND       M01911	// T)¡ío¨¬I
OR LOAD
OUT       P00126	// -
// ========== L_3rd MANDREL SPANKING FWD/BWD ==========
; L229
LOAD      M11080	// L_3rd MAND CYCLE RUN
AND       M1101C	// -
OR        M1136A
OR        M11142
AND NOT   M1101F	// -
AND NOT   M11067	// L_3rd BTM ROT R ORIGIN->
AND NOT   M0067D	// L_3rd SPANKING FWD/BWD SN ALARM
AND NOT   M11368
OUT       M11142
; L232
LOAD      M11142
LOAD      F00094
AND       M01913
OR LOAD
OUT       P0011C	// -
// ========== 06_L_3rd ROTATE Y ==========
; L235
LOAD      M11080	// L_3rd MAND CYCLE RUN
AND       M11020	// -
AND NOT   M04060	// -
LOAD      M10812	// T)L_2nd ROT Y MANDREL POS ->
AND       M01562	// L_3rd SPK Y HOME COMPLETE
OR LOAD
OR        M03060	// -
AND       T0706	// L_3rd SPK Y READY 2s
OUT       M03060	// -

